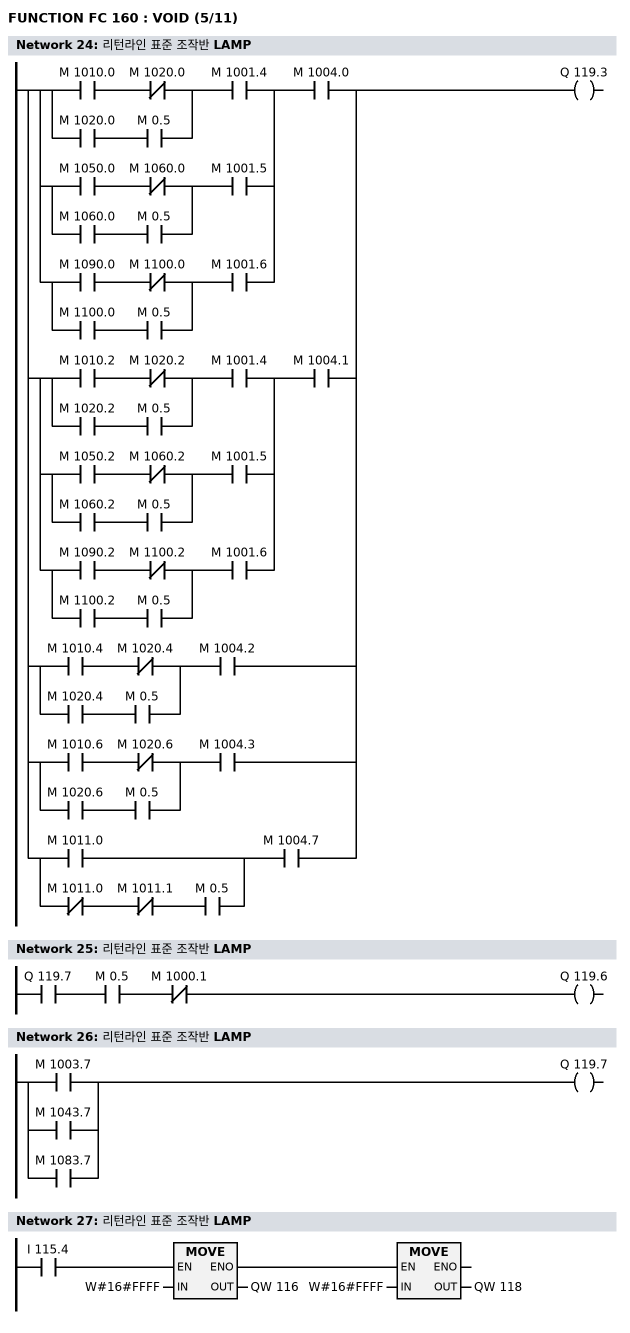

      A(    ;
      A(    ;
      A     M   1010.0;
      AN    M   1020.0;
      O     ;
      A     M   1020.0;
      A     M      0.5;
      )     ;
      A     M   1001.4;
      O     ;
      A(    ;
      A     M   1050.0;
      AN    M   1060.0;
      O     ;
      A     M   1060.0;
      A     M      0.5;
      )     ;
      A     M   1001.5;
      O     ;
      A(    ;
      A     M   1090.0;
      AN    M   1100.0;
      O     ;
      A     M   1100.0;
      A     M      0.5;
      )     ;
      A     M   1001.6;
      )     ;
      A     M   1004.0;
      O     ;
      A(    ;
      A(    ;
      A     M   1010.2;
      AN    M   1020.2;
      O     ;
      A     M   1020.2;
      A     M      0.5;
      )     ;
      A     M   1001.4;
      O     ;
      A(    ;
      A     M   1050.2;
      AN    M   1060.2;
      O     ;
      A     M   1060.2;
      A     M      0.5;
      )     ;
      A     M   1001.5;
      O     ;
      A(    ;
      A     M   1090.2;
      AN    M   1100.2;
      O     ;
      A     M   1100.2;
      A     M      0.5;
      )     ;
      A     M   1001.6;
      )     ;
      A     M   1004.1;
      O     ;
      A(    ;
      A     M   1010.4;
      AN    M   1020.4;
      O     ;
      A     M   1020.4;
      A     M      0.5;
      )     ;
      A     M   1004.2;
      O     ;
      A(    ;
      A     M   1010.6;
      AN    M   1020.6;
      O     ;
      A     M   1020.6;
      A     M      0.5;
      )     ;
      A     M   1004.3;
      O     ;
      A(    ;
      O     M   1011.0;
      O     ;
      AN    M   1011.0;
      AN    M   1011.1;
      A     M      0.5;
      )     ;
      A     M   1004.7;
      =     Q    119.3;
NETWORK
TITLE =리턴라인 표준 조작반 LAMP

      A     Q    119.7;
      A     M      0.5;
      AN    M   1000.1;
      =     Q    119.6;
NETWORK
TITLE =리턴라인 표준 조작반 LAMP

      O     M   1003.7;
      O     M   1043.7;
      O     M   1083.7;
      =     Q    119.7;
NETWORK
TITLE =리턴라인 표준 조작반 LAMP

      A(    ;
      A     I    115.4;
      JNB   _001;
      L     W#16#FFFF;
      T     QW   116;
      SET   ;
      SAVE  ;
      CLR   ;
_001: A     BR;
      )     ;
      JNB   _002;
      L     W#16#FFFF;
      T     QW   118;
_002: NOP   0;
NETWORK
TITLE =리턴라인 표준 조작반 LAMP
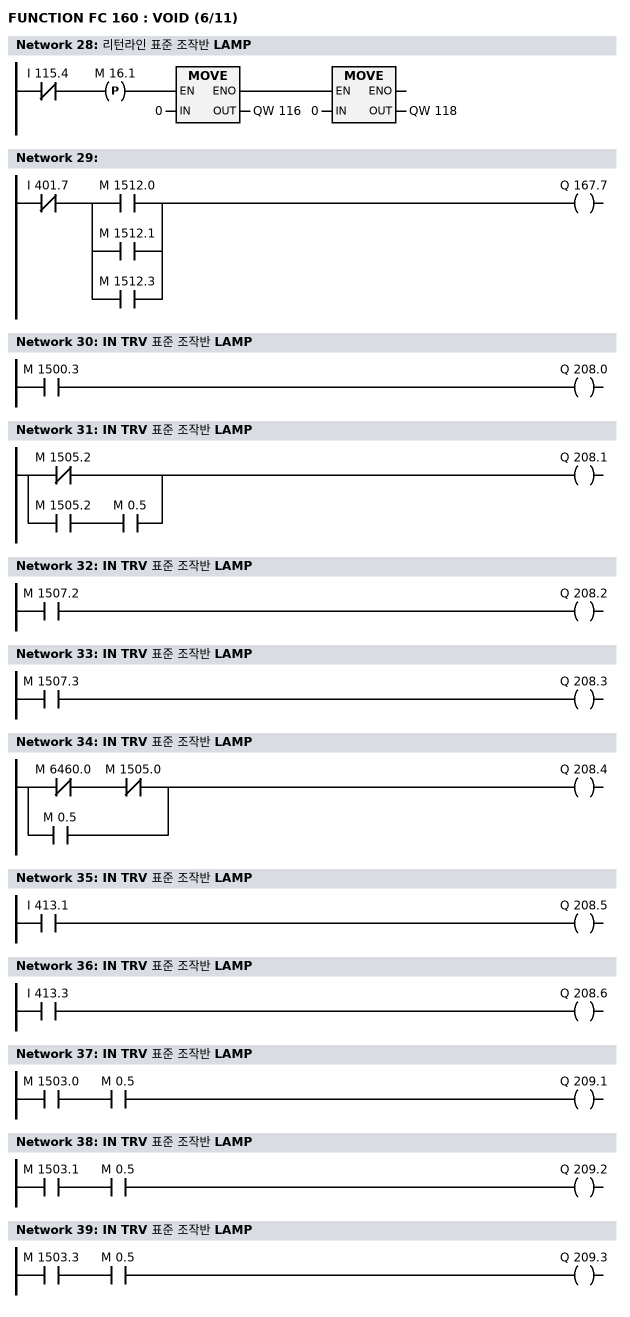

      A(    ;
      AN    I    115.4;
      FP    M     16.1;
      JNB   _003;
      L     0;
      T     QW   116;
      SET   ;
      SAVE  ;
      CLR   ;
_003: A     BR;
      )     ;
      JNB   _004;
      L     0;
      T     QW   118;
_004: NOP   0;
NETWORK
TITLE =

      AN    I    401.7;
      A(    ;
      O     M   1512.0;
      O     M   1512.1;
      O     M   1512.3;
      )     ;
      =     Q    167.7;
NETWORK
TITLE =IN TRV 표준 조작반 LAMP

      A     M   1500.3;
      =     Q    208.0;
NETWORK
TITLE =IN TRV 표준 조작반 LAMP

      ON    M   1505.2;
      O     ;
      A     M   1505.2;
      A     M      0.5;
      =     Q    208.1;
NETWORK
TITLE =IN TRV 표준 조작반 LAMP

      A     M   1507.2;
      =     Q    208.2;
NETWORK
TITLE =IN TRV 표준 조작반 LAMP

      A     M   1507.3;
      =     Q    208.3;
NETWORK
TITLE =IN TRV 표준 조작반 LAMP

      AN    M   6460.0;
      AN    M   1505.0;
      O     M      0.5;
      =     Q    208.4;
NETWORK
TITLE =IN TRV 표준 조작반 LAMP

      A     I    413.1;
      =     Q    208.5;
NETWORK
TITLE =IN TRV 표준 조작반 LAMP

      A     I    413.3;
      =     Q    208.6;
NETWORK
TITLE =IN TRV 표준 조작반 LAMP

      A     M   1503.0;
      A     M      0.5;
      =     Q    209.1;
NETWORK
TITLE =IN TRV 표준 조작반 LAMP

      A     M   1503.1;
      A     M      0.5;
      =     Q    209.2;
NETWORK
TITLE =IN TRV 표준 조작반 LAMP

      A     M   1503.3;
      A     M      0.5;
      =     Q    209.3;
NETWORK
TITLE =IN TRV 표준 조작반 LAMP
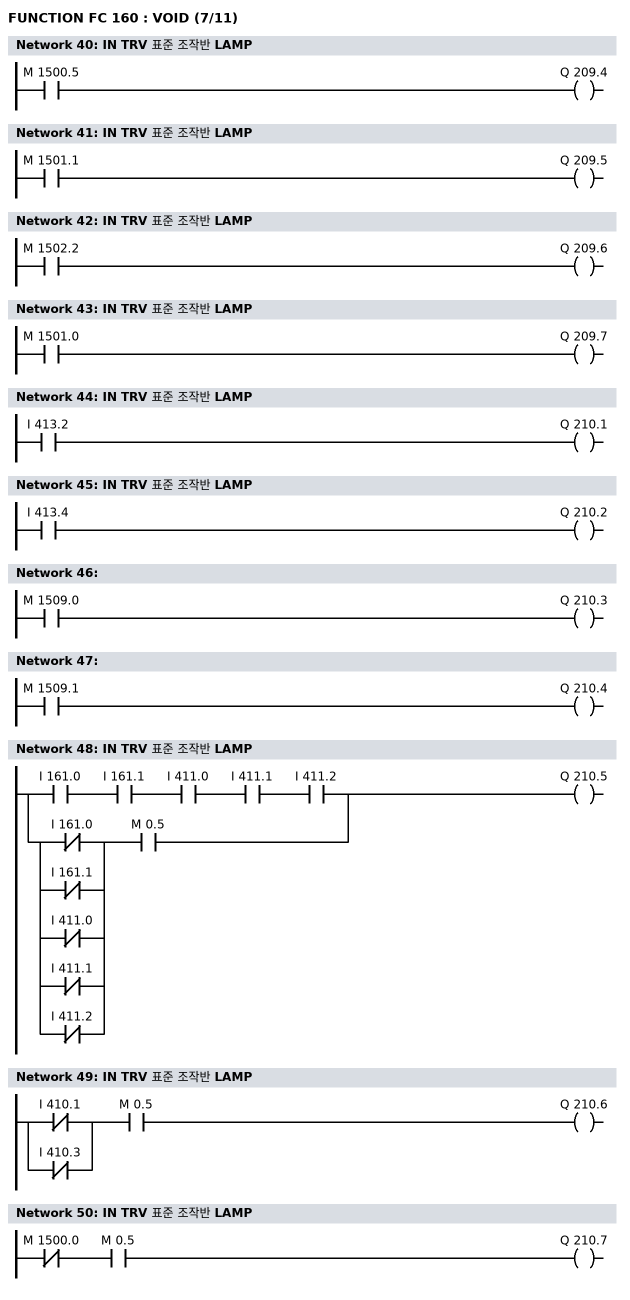

      A     M   1500.5;
      =     Q    209.4;
NETWORK
TITLE =IN TRV 표준 조작반 LAMP

      A     M   1501.1;
      =     Q    209.5;
NETWORK
TITLE =IN TRV 표준 조작반 LAMP

      A     M   1502.2;
      =     Q    209.6;
NETWORK
TITLE =IN TRV 표준 조작반 LAMP

      A     M   1501.0;
      =     Q    209.7;
NETWORK
TITLE =IN TRV 표준 조작반 LAMP

      A     I    413.2;
      =     Q    210.1;
NETWORK
TITLE =IN TRV 표준 조작반 LAMP

      A     I    413.4;
      =     Q    210.2;
NETWORK
TITLE =

      A     M   1509.0;
      =     Q    210.3;
NETWORK
TITLE =

      A     M   1509.1;
      =     Q    210.4;
NETWORK
TITLE =IN TRV 표준 조작반 LAMP

      A     I    161.0;
      A     I    161.1;
      A     I    411.0;
      A     I    411.1;
      A     I    411.2;
      O     ;
      A(    ;
      ON    I    161.0;
      ON    I    161.1;
      ON    I    411.0;
      ON    I    411.1;
      ON    I    411.2;
      )     ;
      A     M      0.5;
      =     Q    210.5;
NETWORK
TITLE =IN TRV 표준 조작반 LAMP

      A(    ;
      ON    I    410.1;
      ON    I    410.3;
      )     ;
      A     M      0.5;
      =     Q    210.6;
NETWORK
TITLE =IN TRV 표준 조작반 LAMP

      AN    M   1500.0;
      A     M      0.5;
      =     Q    210.7;
NETWORK
TITLE =IN TRV 표준 조작반 LAMP
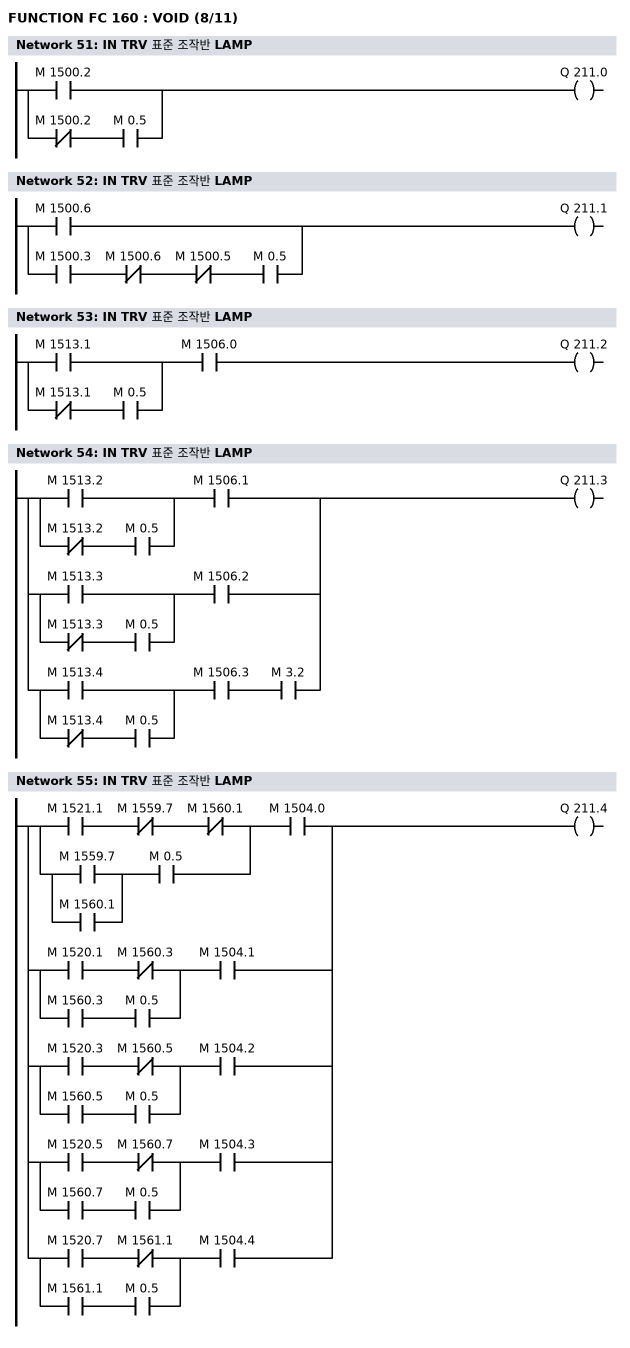

      O     M   1500.2;
      O     ;
      AN    M   1500.2;
      A     M      0.5;
      =     Q    211.0;
NETWORK
TITLE =IN TRV 표준 조작반 LAMP

      O     M   1500.6;
      O     ;
      A     M   1500.3;
      AN    M   1500.6;
      AN    M   1500.5;
      A     M      0.5;
      =     Q    211.1;
NETWORK
TITLE =IN TRV 표준 조작반 LAMP

      A(    ;
      O     M   1513.1;
      O     ;
      AN    M   1513.1;
      A     M      0.5;
      )     ;
      A     M   1506.0;
      =     Q    211.2;
NETWORK
TITLE =IN TRV 표준 조작반 LAMP

      A(    ;
      O     M   1513.2;
      O     ;
      AN    M   1513.2;
      A     M      0.5;
      )     ;
      A     M   1506.1;
      O     ;
      A(    ;
      O     M   1513.3;
      O     ;
      AN    M   1513.3;
      A     M      0.5;
      )     ;
      A     M   1506.2;
      O     ;
      A(    ;
      O     M   1513.4;
      O     ;
      AN    M   1513.4;
      A     M      0.5;
      )     ;
      A     M   1506.3;
      A     M      3.2;
      =     Q    211.3;
NETWORK
TITLE =IN TRV 표준 조작반 LAMP

      A(    ;
      A     M   1521.1;
      AN    M   1559.7;
      AN    M   1560.1;
      O     ;
      A(    ;
      O     M   1559.7;
      O     M   1560.1;
      )     ;
      A     M      0.5;
      )     ;
      A     M   1504.0;
      O     ;
      A(    ;
      A     M   1520.1;
      AN    M   1560.3;
      O     ;
      A     M   1560.3;
      A     M      0.5;
      )     ;
      A     M   1504.1;
      O     ;
      A(    ;
      A     M   1520.3;
      AN    M   1560.5;
      O     ;
      A     M   1560.5;
      A     M      0.5;
      )     ;
      A     M   1504.2;
      O     ;
      A(    ;
      A     M   1520.5;
      AN    M   1560.7;
      O     ;
      A     M   1560.7;
      A     M      0.5;
      )     ;
      A     M   1504.3;
      O     ;
      A(    ;
      A     M   1520.7;
      AN    M   1561.1;
      O     ;
      A     M   1561.1;
      A     M      0.5;
      )     ;
      A     M   1504.4;
      =     Q    211.4;
NETWORK
TITLE =IN TRV 표준 조작반 LAMP
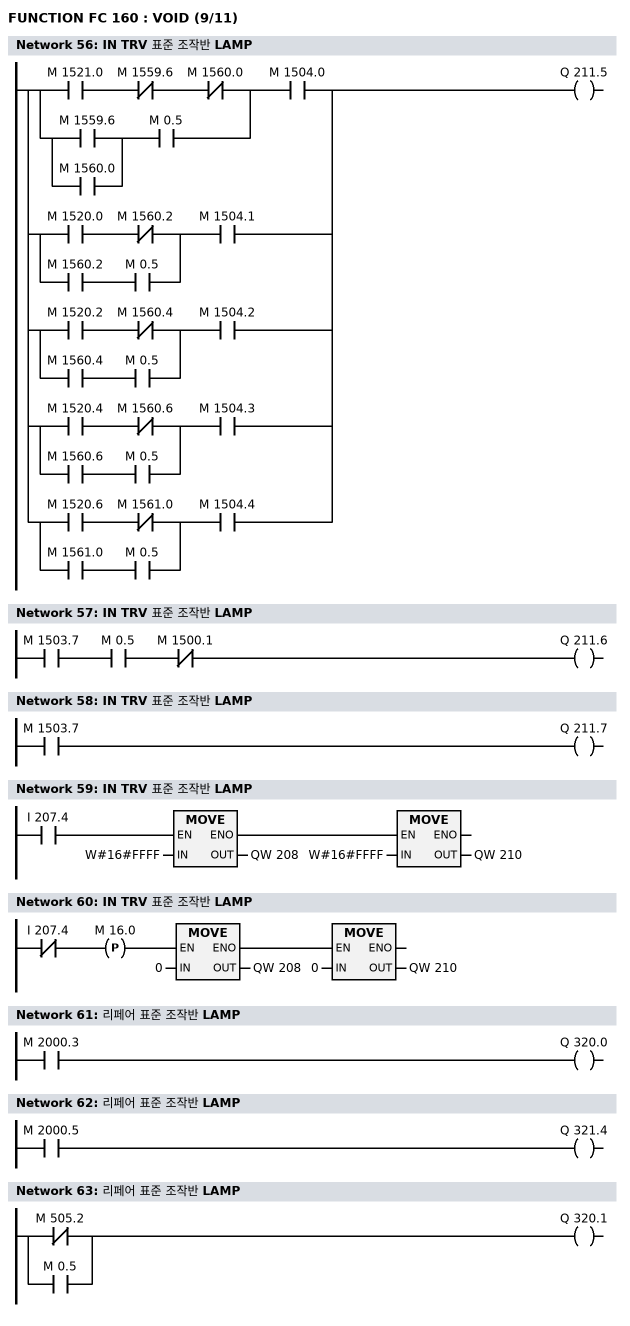

      A(    ;
      A     M   1521.0;
      AN    M   1559.6;
      AN    M   1560.0;
      O     ;
      A(    ;
      O     M   1559.6;
      O     M   1560.0;
      )     ;
      A     M      0.5;
      )     ;
      A     M   1504.0;
      O     ;
      A(    ;
      A     M   1520.0;
      AN    M   1560.2;
      O     ;
      A     M   1560.2;
      A     M      0.5;
      )     ;
      A     M   1504.1;
      O     ;
      A(    ;
      A     M   1520.2;
      AN    M   1560.4;
      O     ;
      A     M   1560.4;
      A     M      0.5;
      )     ;
      A     M   1504.2;
      O     ;
      A(    ;
      A     M   1520.4;
      AN    M   1560.6;
      O     ;
      A     M   1560.6;
      A     M      0.5;
      )     ;
      A     M   1504.3;
      O     ;
      A(    ;
      A     M   1520.6;
      AN    M   1561.0;
      O     ;
      A     M   1561.0;
      A     M      0.5;
      )     ;
      A     M   1504.4;
      =     Q    211.5;
NETWORK
TITLE =IN TRV 표준 조작반 LAMP

      A     M   1503.7;
      A     M      0.5;
      AN    M   1500.1;
      =     Q    211.6;
NETWORK
TITLE =IN TRV 표준 조작반 LAMP

      A     M   1503.7;
      =     Q    211.7;
NETWORK
TITLE =IN TRV 표준 조작반 LAMP

      A(    ;
      A     I    207.4;
      JNB   _005;
      L     W#16#FFFF;
      T     QW   208;
      SET   ;
      SAVE  ;
      CLR   ;
_005: A     BR;
      )     ;
      JNB   _006;
      L     W#16#FFFF;
      T     QW   210;
_006: NOP   0;
NETWORK
TITLE =IN TRV 표준 조작반 LAMP

      A(    ;
      AN    I    207.4;
      FP    M     16.0;
      JNB   _007;
      L     0;
      T     QW   208;
      SET   ;
      SAVE  ;
      CLR   ;
_007: A     BR;
      )     ;
      JNB   _008;
      L     0;
      T     QW   210;
_008: NOP   0;
NETWORK
TITLE =리페어 표준 조작반 LAMP

      A     M   2000.3;
      =     Q    320.0;
NETWORK
TITLE =리페어 표준 조작반 LAMP

      A     M   2000.5;
      =     Q    321.4;
NETWORK
TITLE =리페어 표준 조작반 LAMP

      ON    M    505.2;
      O     M      0.5;
      =     Q    320.1;
NETWORK
TITLE =리페어 표준 조작반 LAMP
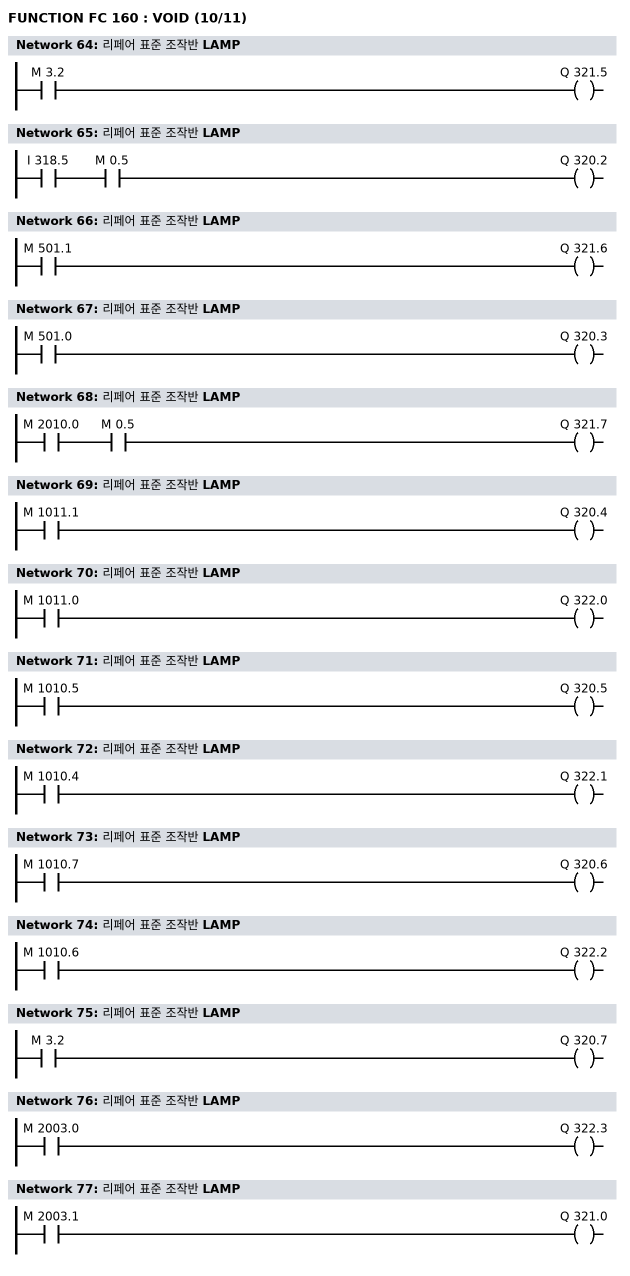

      A     M      3.2;
      =     Q    321.5;
NETWORK
TITLE =리페어 표준 조작반 LAMP

      A     I    318.5;
      A     M      0.5;
      =     Q    320.2;
NETWORK
TITLE =리페어 표준 조작반 LAMP

      A     M    501.1;
      =     Q    321.6;
NETWORK
TITLE =리페어 표준 조작반 LAMP

      A     M    501.0;
      =     Q    320.3;
NETWORK
TITLE =리페어 표준 조작반 LAMP

      A     M   2010.0;
      A     M      0.5;
      =     Q    321.7;
NETWORK
TITLE =리페어 표준 조작반 LAMP

      A     M   1011.1;
      =     Q    320.4;
NETWORK
TITLE =리페어 표준 조작반 LAMP

      A     M   1011.0;
      =     Q    322.0;
NETWORK
TITLE =리페어 표준 조작반 LAMP

      A     M   1010.5;
      =     Q    320.5;
NETWORK
TITLE =리페어 표준 조작반 LAMP

      A     M   1010.4;
      =     Q    322.1;
NETWORK
TITLE =리페어 표준 조작반 LAMP

      A     M   1010.7;
      =     Q    320.6;
NETWORK
TITLE =리페어 표준 조작반 LAMP

      A     M   1010.6;
      =     Q    322.2;
NETWORK
TITLE =리페어 표준 조작반 LAMP

      A     M      3.2;
      =     Q    320.7;
NETWORK
TITLE =리페어 표준 조작반 LAMP

      A     M   2003.0;
      =     Q    322.3;
NETWORK
TITLE =리페어 표준 조작반 LAMP

      A     M   2003.1;
      =     Q    321.0;
NETWORK
TITLE =리페어 표준 조작반 LAMP
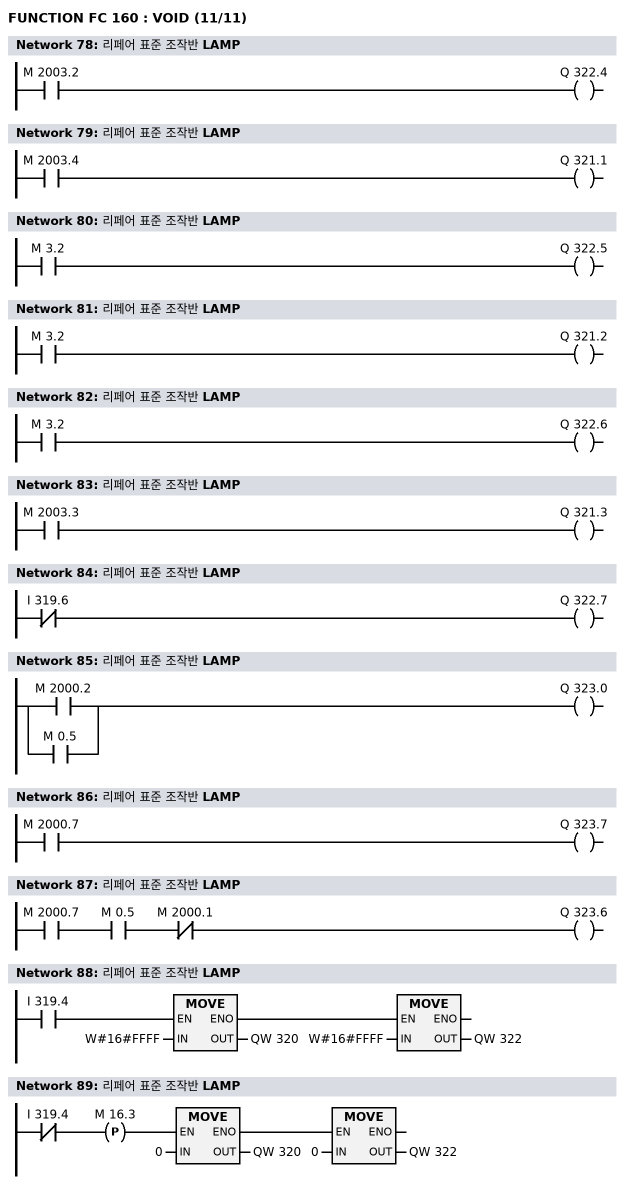

      A     M   2003.2;
      =     Q    322.4;
NETWORK
TITLE =리페어 표준 조작반 LAMP

      A     M   2003.4;
      =     Q    321.1;
NETWORK
TITLE =리페어 표준 조작반 LAMP

      A     M      3.2;
      =     Q    322.5;
NETWORK
TITLE =리페어 표준 조작반 LAMP

      A     M      3.2;
      =     Q    321.2;
NETWORK
TITLE =리페어 표준 조작반 LAMP

      A     M      3.2;
      =     Q    322.6;
NETWORK
TITLE =리페어 표준 조작반 LAMP

      A     M   2003.3;
      =     Q    321.3;
NETWORK
TITLE =리페어 표준 조작반 LAMP

      AN    I    319.6;
      =     Q    322.7;
NETWORK
TITLE =리페어 표준 조작반 LAMP

      O     M   2000.2;
      O     M      0.5;
      =     Q    323.0;
NETWORK
TITLE =리페어 표준 조작반 LAMP

      A     M   2000.7;
      =     Q    323.7;
NETWORK
TITLE =리페어 표준 조작반 LAMP

      A     M   2000.7;
      A     M      0.5;
      AN    M   2000.1;
      =     Q    323.6;
NETWORK
TITLE =리페어 표준 조작반 LAMP

      A(    ;
      A     I    319.4;
      JNB   _009;
      L     W#16#FFFF;
      T     QW   320;
      SET   ;
      SAVE  ;
      CLR   ;
_009: A     BR;
      )     ;
      JNB   _00a;
      L     W#16#FFFF;
      T     QW   322;
_00a: NOP   0;
NETWORK
TITLE =리페어 표준 조작반 LAMP

      A(    ;
      AN    I    319.4;
      FP    M     16.3;
      JNB   _00b;
      L     0;
      T     QW   320;
      SET   ;
      SAVE  ;
      CLR   ;
_00b: A     BR;
      )     ;
      JNB   _00c;
      L     0;
      T     QW   322;
_00c: NOP   0;
END_FUNCTION

FUNCTION FC 324 : VOID
TITLE =
VERSION : 0.1

BEGIN
NETWORK
TITLE =
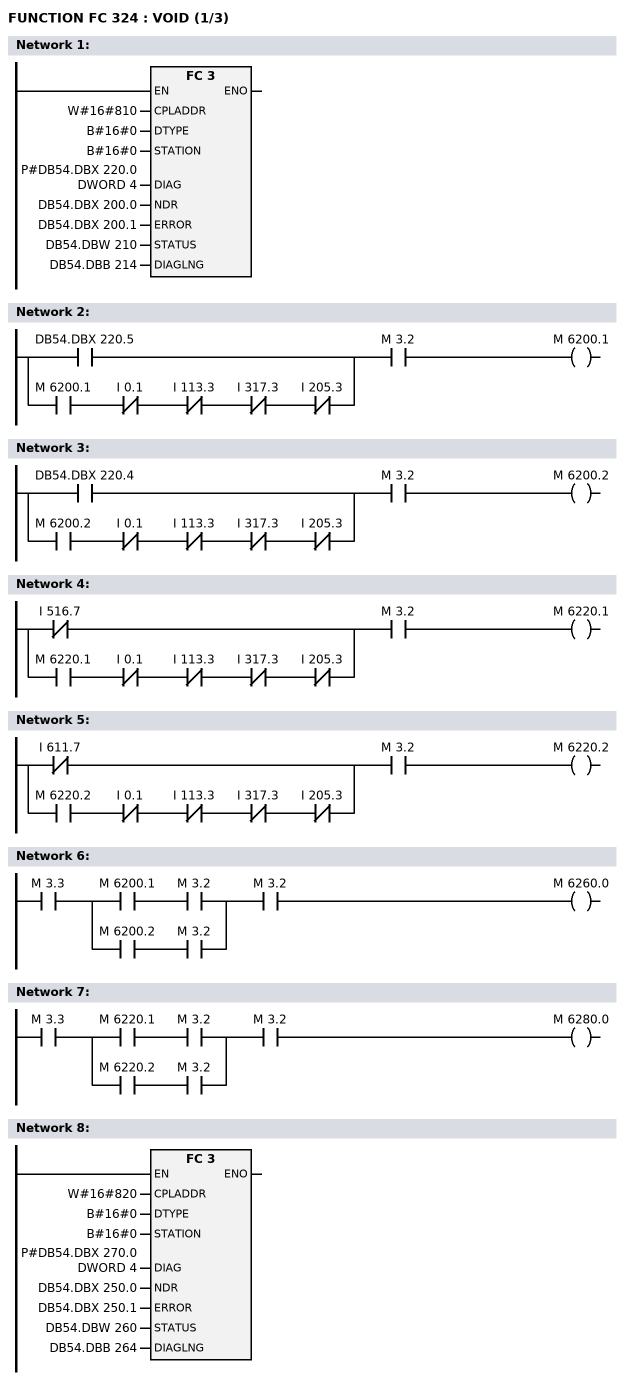

      CALL FC     3 (
           CPLADDR                  := W#16#810,
           DTYPE                    := B#16#0,
           STATION                  := B#16#0,
           DIAG                     := P#DB54.DBX 220.0 DWORD 4,
           NDR                      := DB54.DBX  200.0,
           ERROR                    := DB54.DBX  200.1,
           STATUS                   := DB54.DBW  210,
           DIAGLNG                  := DB54.DBB  214);
      NOP   0;
NETWORK
TITLE =

      A(    ;
      O     DB54.DBX  220.5;
      O     ;
      A     M   6200.1;
      AN    I      0.1;
      AN    I    113.3;
      AN    I    317.3;
      AN    I    205.3;
      )     ;
      A     M      3.2;
      =     M   6200.1;
NETWORK
TITLE =

      A(    ;
      O     DB54.DBX  220.4;
      O     ;
      A     M   6200.2;
      AN    I      0.1;
      AN    I    113.3;
      AN    I    317.3;
      AN    I    205.3;
      )     ;
      A     M      3.2;
      =     M   6200.2;
NETWORK
TITLE =

      A(    ;
      ON    I    516.7;
      O     ;
      A     M   6220.1;
      AN    I      0.1;
      AN    I    113.3;
      AN    I    317.3;
      AN    I    205.3;
      )     ;
      A     M      3.2;
      =     M   6220.1;
NETWORK
TITLE =

      A(    ;
      ON    I    611.7;
      O     ;
      A     M   6220.2;
      AN    I      0.1;
      AN    I    113.3;
      AN    I    317.3;
      AN    I    205.3;
      )     ;
      A     M      3.2;
      =     M   6220.2;
NETWORK
TITLE =

      A     M      3.3;
      A(    ;
      A     M   6200.1;
      A     M      3.2;
      O     ;
      A     M   6200.2;
      A     M      3.2;
      )     ;
      A     M      3.2;
      =     M   6260.0;
NETWORK
TITLE =

      A     M      3.3;
      A(    ;
      A     M   6220.1;
      A     M      3.2;
      O     ;
      A     M   6220.2;
      A     M      3.2;
      )     ;
      A     M      3.2;
      =     M   6280.0;
NETWORK
TITLE =

      CALL FC     3 (
           CPLADDR                  := W#16#820,
           DTYPE                    := B#16#0,
           STATION                  := B#16#0,
           DIAG                     := P#DB54.DBX 270.0 DWORD 4,
           NDR                      := DB54.DBX  250.0,
           ERROR                    := DB54.DBX  250.1,
           STATUS                   := DB54.DBW  260,
           DIAGLNG                  := DB54.DBB  264);
      NOP   0;
NETWORK
TITLE =
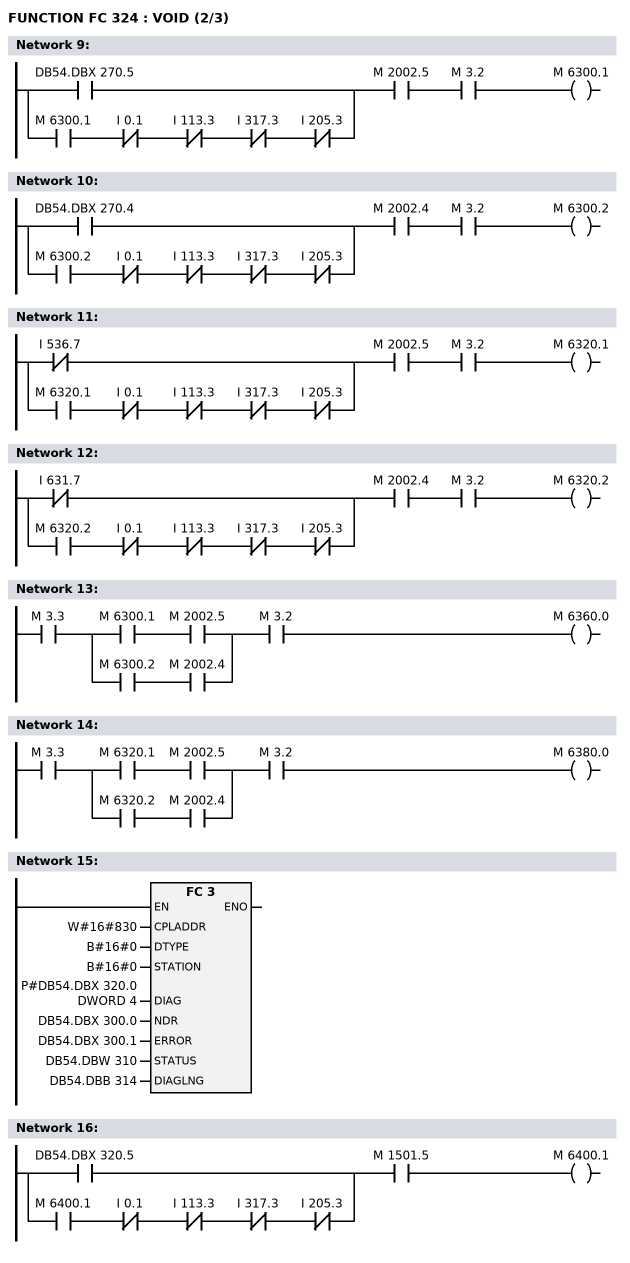

      A(    ;
      O     DB54.DBX  270.5;
      O     ;
      A     M   6300.1;
      AN    I      0.1;
      AN    I    113.3;
      AN    I    317.3;
      AN    I    205.3;
      )     ;
      A     M   2002.5;
      A     M      3.2;
      =     M   6300.1;
NETWORK
TITLE =

      A(    ;
      O     DB54.DBX  270.4;
      O     ;
      A     M   6300.2;
      AN    I      0.1;
      AN    I    113.3;
      AN    I    317.3;
      AN    I    205.3;
      )     ;
      A     M   2002.4;
      A     M      3.2;
      =     M   6300.2;
NETWORK
TITLE =

      A(    ;
      ON    I    536.7;
      O     ;
      A     M   6320.1;
      AN    I      0.1;
      AN    I    113.3;
      AN    I    317.3;
      AN    I    205.3;
      )     ;
      A     M   2002.5;
      A     M      3.2;
      =     M   6320.1;
NETWORK
TITLE =

      A(    ;
      ON    I    631.7;
      O     ;
      A     M   6320.2;
      AN    I      0.1;
      AN    I    113.3;
      AN    I    317.3;
      AN    I    205.3;
      )     ;
      A     M   2002.4;
      A     M      3.2;
      =     M   6320.2;
NETWORK
TITLE =

      A     M      3.3;
      A(    ;
      A     M   6300.1;
      A     M   2002.5;
      O     ;
      A     M   6300.2;
      A     M   2002.4;
      )     ;
      A     M      3.2;
      =     M   6360.0;
NETWORK
TITLE =

      A     M      3.3;
      A(    ;
      A     M   6320.1;
      A     M   2002.5;
      O     ;
      A     M   6320.2;
      A     M   2002.4;
      )     ;
      A     M      3.2;
      =     M   6380.0;
NETWORK
TITLE =

      CALL FC     3 (
           CPLADDR                  := W#16#830,
           DTYPE                    := B#16#0,
           STATION                  := B#16#0,
           DIAG                     := P#DB54.DBX 320.0 DWORD 4,
           NDR                      := DB54.DBX  300.0,
           ERROR                    := DB54.DBX  300.1,
           STATUS                   := DB54.DBW  310,
           DIAGLNG                  := DB54.DBB  314);
      NOP   0;
NETWORK
TITLE =

      A(    ;
      O     DB54.DBX  320.5;
      O     ;
      A     M   6400.1;
      AN    I      0.1;
      AN    I    113.3;
      AN    I    317.3;
      AN    I    205.3;
      )     ;
      A     M   1501.5;
      =     M   6400.1;
NETWORK
TITLE =
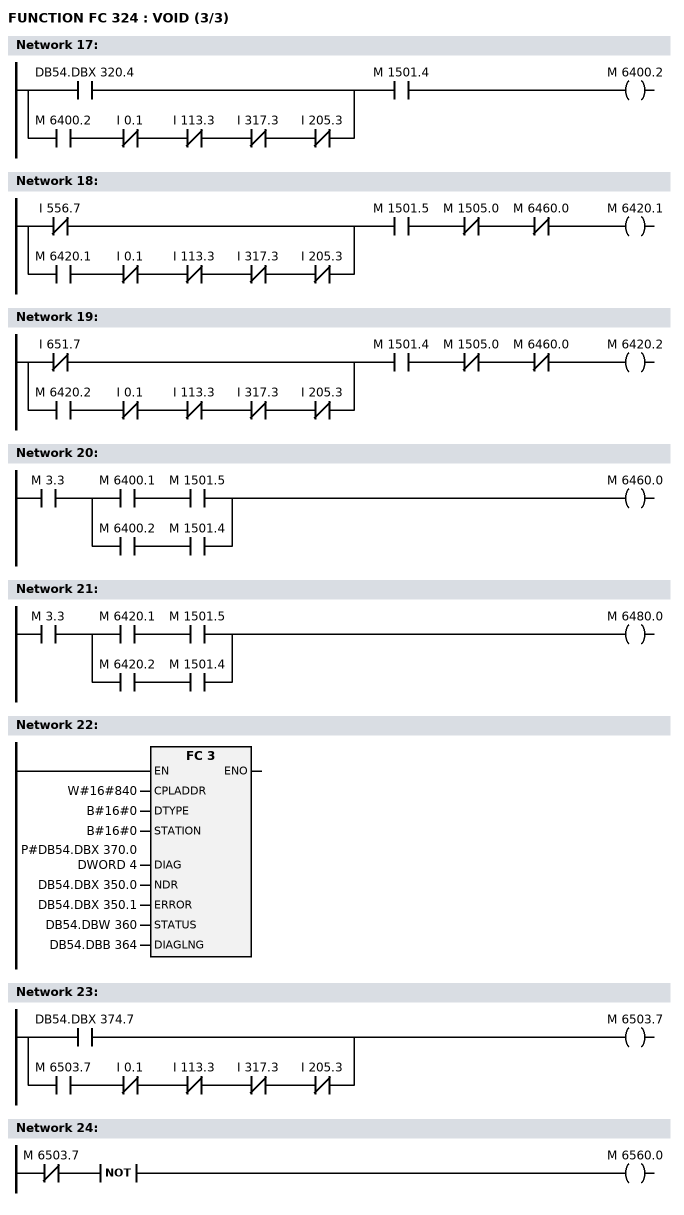

      A(    ;
      O     DB54.DBX  320.4;
      O     ;
      A     M   6400.2;
      AN    I      0.1;
      AN    I    113.3;
      AN    I    317.3;
      AN    I    205.3;
      )     ;
      A     M   1501.4;
      =     M   6400.2;
NETWORK
TITLE =

      A(    ;
      ON    I    556.7;
      O     ;
      A     M   6420.1;
      AN    I      0.1;
      AN    I    113.3;
      AN    I    317.3;
      AN    I    205.3;
      )     ;
      A     M   1501.5;
      AN    M   1505.0;
      AN    M   6460.0;
      =     M   6420.1;
NETWORK
TITLE =

      A(    ;
      ON    I    651.7;
      O     ;
      A     M   6420.2;
      AN    I      0.1;
      AN    I    113.3;
      AN    I    317.3;
      AN    I    205.3;
      )     ;
      A     M   1501.4;
      AN    M   1505.0;
      AN    M   6460.0;
      =     M   6420.2;
NETWORK
TITLE =

      A     M      3.3;
      A(    ;
      A     M   6400.1;
      A     M   1501.5;
      O     ;
      A     M   6400.2;
      A     M   1501.4;
      )     ;
      =     M   6460.0;
NETWORK
TITLE =

      A     M      3.3;
      A(    ;
      A     M   6420.1;
      A     M   1501.5;
      O     ;
      A     M   6420.2;
      A     M   1501.4;
      )     ;
      =     M   6480.0;
NETWORK
TITLE =

      CALL FC     3 (
           CPLADDR                  := W#16#840,
           DTYPE                    := B#16#0,
           STATION                  := B#16#0,
           DIAG                     := P#DB54.DBX 370.0 DWORD 4,
           NDR                      := DB54.DBX  350.0,
           ERROR                    := DB54.DBX  350.1,
           STATUS                   := DB54.DBW  360,
           DIAGLNG                  := DB54.DBB  364);
      NOP   0;
NETWORK
TITLE =

      O     DB54.DBX  374.7;
      O     ;
      A     M   6503.7;
      AN    I      0.1;
      AN    I    113.3;
      AN    I    317.3;
      AN    I    205.3;
      =     M   6503.7;
NETWORK
TITLE =

      AN    M   6503.7;
      NOT   ;
      =     M   6560.0;
END_FUNCTION

FUNCTION_BLOCK FB 406
TITLE =Data Block Move Program
AUTHOR : HMC
FAMILY : Car_Type
NAME : Car_Type
VERSION : 1.0


VAR_INPUT
  FWD_Pulse : BOOL ;
  RET_Pulse : BOOL ;
  Source_DB : INT ;
  Start_Add : INT ;
  Stn_Amount : INT ;
  Byte_per_Stn : INT ;
  Cpu_Run_Pulse : BOOL ;
END_VAR
VAR_OUTPUT
  Complete : BOOL ;
END_VAR
VAR
  Operation : BOOL ;
  Mask_Arr : ARRAY  [0 .. 599 ] OF BYTE ;
  Ret : INT ;
  Data_Type : WORD ;
  Data_Length : INT ;
  Secend_Stn_Add : INT ;
  Fill_Source : WORD ;
END_VAR
VAR_TEMP
  First_Stn : ANY ;
  Mask : ANY ;
  Second_Stn : ANY ;
  Save_AR1 : DWORD ;
  Save_AR2 : DWORD ;
  Save_DB : INT ;
  Save_DI : INT ;
  First_Stn_1 : ANY ;
END_VAR
BEGIN
NETWORK
TITLE =Save adress register and DB's

      TAR1  #Save_AR1; // Save adress register 1
      TAR2  #Save_AR2; // Save adress register 2
      L     DBNO; // loads the number of the shared open data block
      T     #Save_DB;
      L     DINO; // loads the number of the opened instance data block
      T     #Save_DI;
NETWORK
TITLE =Operation Pulse

      O     #FWD_Pulse; // External ForwardOperation Signal
      O     #RET_Pulse; // External Return Operation Signal
      FP    #Operation; // Operation Pulse
      JNB   _End; // Jump to End
NETWORK
TITLE =Data Type Select In ANY Type Parameter

      A(    ; // If Source DB is Not Zero
      L     #Source_DB;
      L     0;
      <>I   ;
      )     ;
      JNB   _001; // Jump to Next Step
      L     W#16#8400; // Load "8400" _ Means "DB Area"
      T     #Data_Type; // Transfer to Data_Type
_001: NOP   0;
NETWORK
TITLE =Data Type Select In ANY Type Parameter

      A(    ; // If DB_NO is Zero
      L     #Source_DB;
      L     0;
      ==I   ;
      )     ;
      JNB   _002; // Jump to Next Step
      L     W#16#8300; // Load "8300" _ Means "Bit Memory Area"
      T     #Data_Type; // Transfer to Data_Type
_002: NOP   0;
NETWORK
TITLE =Data Length Select

      L     #Stn_Amount; // Station Amount - 1
      L     1;
      -I    ;
      L     #Byte_per_Stn; // Multi Length Per Station
      *I    ;
      T     #Data_Length; // Transfer to Data Length
NETWORK
TITLE =2nd Station Address Select

      L     #Start_Add; // Pluse Start Address And Length
      L     #Byte_per_Stn;
      +I    ;
      T     #Secend_Stn_Add; // Transfer to Second Station Address
NETWORK
TITLE =Make a "ANY" Type Data

      LAR1  P##First_Stn; // Load 1st Station Address of ANY Pointer In "AR1"

      L     B#16#10; // Load Syntax ID For S7 "10"
      T     LB [AR1,P#0.0]; // Transfer ID to the ANY Pointer

      L     B#16#2; // Load Data Type _ "2" means "BYTE"
      T     LB [AR1,P#1.0]; // Transfer Data Type to the ANY Pointer

      L     #Data_Length; // Load the Length of Source Data
      T     LW [AR1,P#2.0]; // Transfer the Numbers to the ANY Pointer

      L     #Source_DB; // Load DB Number _ "0" means don't use "DB"
      T     LW [AR1,P#4.0]; // Transfer the Numbers to the ANY Pointer

      L     #Data_Type; // Load Data Type _ "83" means "Bit Memory" Area
      T     LW [AR1,P#6.0]; //                  "84" means "DB" Area

      L     #Start_Add; // Load Start Address
      SLW   3; // Shift Left Word _ "3" Bit
      T     LW [AR1,P#8.0]; // Transfer the Address to the ANY Pointer

      LAR1  P##Mask; // Load 2nd Station Address of ANY Pointer In "AR1"

      L     B#16#10; //Load Syntax ID For S7 "10"
      T     LB [AR1,P#0.0]; //Load Syntax ID For S7 "10"

      L     B#16#2; //  Load Data Type _ "2" means "BYTE"
      T     LB [AR1,P#1.0]; // Transfer Data Type to the ANY Pointer

      L     #Data_Length; // Load the Length of Target Data
      T     LW [AR1,P#2.0]; // Transfer the Numbers to the ANY Pointer

      L     #Save_DI; // Load DB Number _ "0" means don't use "DB"
      T     LW [AR1,P#4.0]; // Transfer the Numbers to the ANY Pointer

      L     #Data_Type; // Load Data Type _ "83" means "Bit Memory" Area
      T     LW [AR1,P#6.0]; //                  "84" means "DB" Area

      L     16; //  Load Start Address
      SLW   3; // Shift Left Word _ "3" Bit
      T     LW [AR1,P#8.0]; // Transfer the Address to the ANY Pointer

NETWORK
TITLE =Make a "ANY" Type Data

      LAR1  P##Second_Stn; // Load 1st Station Address of ANY Pointer In "AR1"

      L     B#16#10; // Load Syntax ID For S7 "10"
      T     LB [AR1,P#0.0]; // Transfer ID to the ANY Pointer

      L     B#16#2; // Load Data Type _ "2" means "BYTE"
      T     LB [AR1,P#1.0]; // Transfer Data Type to the ANY Pointer

      L     #Data_Length; // Load the Length of Source Data
      T     LW [AR1,P#2.0]; // Transfer the Numbers to the ANY Pointer

      L     #Source_DB; // Load DB Number _ "0" means don't use "DB"
      T     LW [AR1,P#4.0]; // Transfer the Numbers to the ANY Pointer

      L     #Data_Type; // Load Data Type _ "83" means "Bit Memory" Area
      T     LW [AR1,P#6.0]; //                  "84" means "DB" Area

      L     #Secend_Stn_Add; // Load Second Station Address
      SLW   3; // Shift Left Word _ "3" Bit
      T     LW [AR1,P#8.0]; // Transfer the Address to the ANY Pointer
NETWORK
TITLE =Reset Car Type Transfer Complete Signal

      O     #FWD_Pulse; // External Forward Operation Signal
      O     #RET_Pulse; // External Return Operation Signal
      R     #Complete; // Reset Complete Signal
NETWORK
TITLE =Make Fill Source Data

      L     0;
      T     #Fill_Source;
NETWORK
TITLE =Fwd Block Move to Mask Area

      A     #FWD_Pulse; // External Forward Operation Signal
      AN    #Complete; // Complete Signal is False
      AN    #Cpu_Run_Pulse;
      JNB   _FWD;
      CALL SFC   20 (
           SRCBLK                   := #First_Stn,
           RET_VAL                  := #Ret,
           DSTBLK                   := #Mask);

NETWORK
TITLE =Clear Source Data Area


      CALL SFC   21 (
           IN0                      := #Fill_Source,// "Zero"
           RET_VAL                  := #Ret,
           OUT1                     := #First_Stn);// Transfer to First Station Area

NETWORK
TITLE =Fwd Block Move to Second Station Area


      CALL SFC   20 (
           SRCBLK                   := #Mask,
           RET_VAL                  := #Ret,
           DSTBLK                   := #Second_Stn);

NETWORK
TITLE =Clear Mask Data Area


      CALL SFC   21 (
           IN0                      := #Fill_Source,// "Zero"
           RET_VAL                  := #Ret,
           OUT1                     := #Mask);// Transfer to Mask Area
_FWD: NOP   0;
NETWORK
TITLE =Rev Block Move to Mask Area

      A     #RET_Pulse; // External Return Operation Signal
      AN    #Complete; // Complete Signal is False
      AN    #Cpu_Run_Pulse;
      JNB   _REV;
      CALL SFC   20 (
           SRCBLK                   := #Second_Stn,
           RET_VAL                  := #Ret,
           DSTBLK                   := #Mask);

NETWORK
TITLE =Clear Source Data Area


      CALL SFC   21 (
           IN0                      := #Fill_Source,// "Zero"
           RET_VAL                  := #Ret,
           OUT1                     := #Second_Stn);// Transfer to Second Station Area

NETWORK
TITLE =Rev Block Move to First Station Area


      CALL SFC   20 (
           SRCBLK                   := #Mask,
           RET_VAL                  := #Ret,
           DSTBLK                   := #First_Stn);

NETWORK
TITLE =Clear Mask Data Area


      CALL SFC   21 (
           IN0                      := #Fill_Source,// "Zero"
           RET_VAL                  := #Ret,
           OUT1                     := #Mask);// Transfer to Mask Area
_REV: NOP   0;
NETWORK
TITLE =Set Complete Signal

      S     #Complete;
_End: NOP   0;
END_FUNCTION_BLOCK

FUNCTION_BLOCK FB 426
TITLE =Sensor Error,Lamp Variables Program
AUTHOR : HMC
FAMILY : Common
NAME : Common
VERSION : 1.0


VAR_INPUT
  Enable_Aux : BOOL ;
  Adv_Amount : INT ;
  Ret_Amount : INT ;
  LS_Adv1 : BOOL ;
  LS_Ret1 : BOOL ;
  LS_Adv2 : BOOL ;
  LS_Ret2 : BOOL ;
  LS_Adv3 : BOOL ;
  LS_Ret3 : BOOL ;
  LS_Adv4 : BOOL ;
  LS_Ret4 : BOOL ;
  LS_Adv5 : BOOL ;
  LS_Ret5 : BOOL ;
  LS_Adv6 : BOOL ;
  LS_Ret6 : BOOL ;
  LS_Adv7 : BOOL ;
  LS_Ret7 : BOOL ;
  LS_Adv8 : BOOL ;
  LS_Ret8 : BOOL ;
  SOL_Adv : BOOL ;
  SOL_Ret : BOOL ;
  M_Ready : BOOL ;
  T_CHK1 : TIME ;
  T_CHK2 : TIME ;
  PB_Lamp_CHK : BOOL ;
  PB_Error_Rst : BOOL ;
  M_FLICK : BOOL ;
END_VAR
VAR_OUTPUT
  M_Adv_Err : BOOL ;
  M_Ret_Err : BOOL ;
  LP_Adv : BOOL ;
  LP_Ret : BOOL ;
  Visu_Adv : WORD ;
  Visu_Ret : WORD ;
END_VAR
VAR
  Error_T1 : SFB 4;
  Error_T2 : SFB 4;
  Adv_End_Aux : BOOL ;
  Ret_End_Aux : BOOL ;
  CHK_Aux1 : BOOL ;
  CHK_Aux2 : BOOL ;
  Error_T1_DN : BOOL ;
  Error_T2_DN : BOOL ;
  Adv_Memo : BOOL ;
  Visu_Adv_Arr : ARRAY  [0 .. 15 ] OF BOOL ;
  Visu_Ret_Arr : ARRAY  [0 .. 15 ] OF BOOL ;
  BLK_Move_Ret : INT ;
  Enable : BOOL ;
  Adv_End : BOOL ;
  Ret_End : BOOL ;
END_VAR
BEGIN
NETWORK
TITLE =
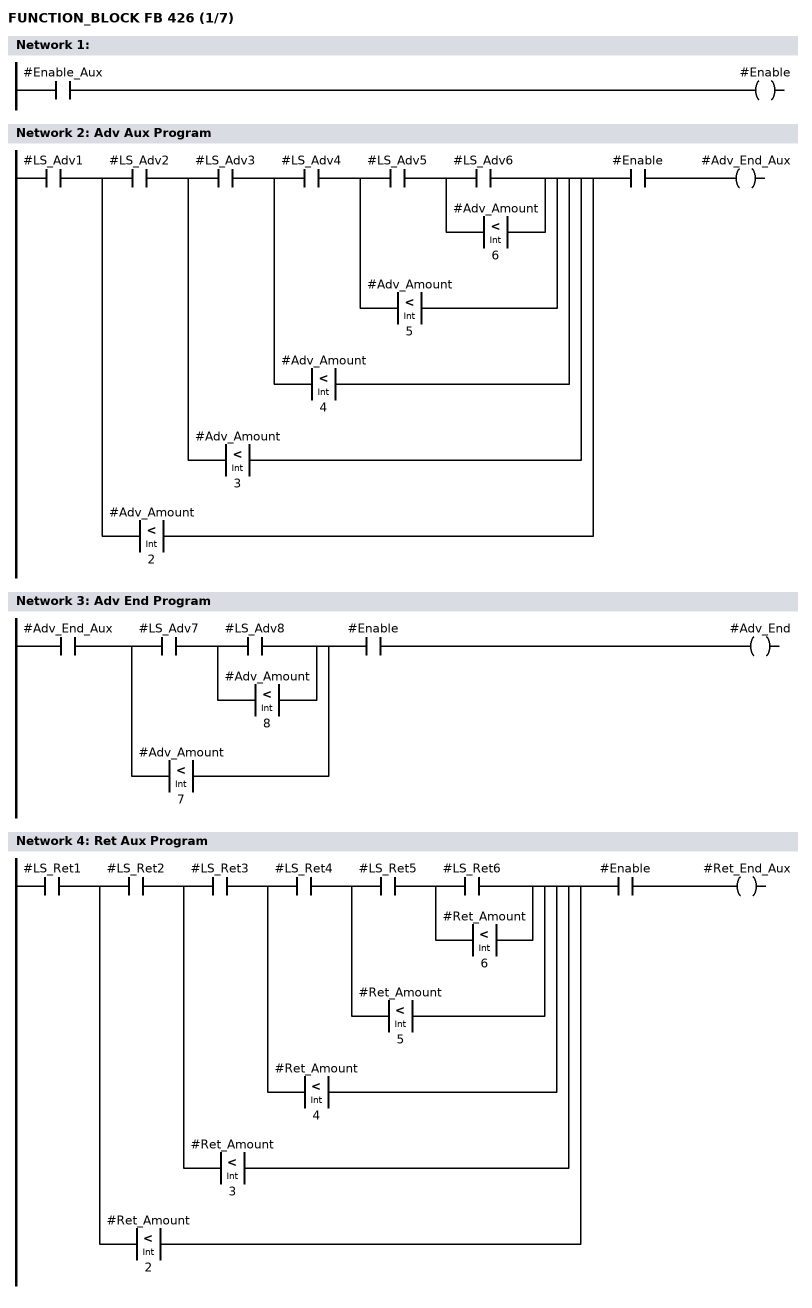

      A     #Enable_Aux;
      =     #Enable;
NETWORK
TITLE =Adv Aux Program

      A     #LS_Adv1;
      A(    ;
      A     #LS_Adv2;
      A(    ;
      A     #LS_Adv3;
      A(    ;
      A     #LS_Adv4;
      A(    ;
      A     #LS_Adv5;
      A(    ;
      O     #LS_Adv6;
      O(    ;
      L     #Adv_Amount;
      L     6;
      <I    ;
      )     ;
      )     ;
      O(    ;
      L     #Adv_Amount;
      L     5;
      <I    ;
      )     ;
      )     ;
      O(    ;
      L     #Adv_Amount;
      L     4;
      <I    ;
      )     ;
      )     ;
      O(    ;
      L     #Adv_Amount;
      L     3;
      <I    ;
      )     ;
      )     ;
      O(    ;
      L     #Adv_Amount;
      L     2;
      <I    ;
      )     ;
      )     ;
      A     #Enable;
      =     #Adv_End_Aux;
NETWORK
TITLE =Adv End Program

      A     #Adv_End_Aux;
      A(    ;
      A     #LS_Adv7;
      A(    ;
      O     #LS_Adv8;
      O(    ;
      L     #Adv_Amount;
      L     8;
      <I    ;
      )     ;
      )     ;
      O(    ;
      L     #Adv_Amount;
      L     7;
      <I    ;
      )     ;
      )     ;
      A     #Enable;
      =     #Adv_End;
NETWORK
TITLE =Ret Aux Program

      A     #LS_Ret1;
      A(    ;
      A     #LS_Ret2;
      A(    ;
      A     #LS_Ret3;
      A(    ;
      A     #LS_Ret4;
      A(    ;
      A     #LS_Ret5;
      A(    ;
      O     #LS_Ret6;
      O(    ;
      L     #Ret_Amount;
      L     6;
      <I    ;
      )     ;
      )     ;
      O(    ;
      L     #Ret_Amount;
      L     5;
      <I    ;
      )     ;
      )     ;
      O(    ;
      L     #Ret_Amount;
      L     4;
      <I    ;
      )     ;
      )     ;
      O(    ;
      L     #Ret_Amount;
      L     3;
      <I    ;
      )     ;
      )     ;
      O(    ;
      L     #Ret_Amount;
      L     2;
      <I    ;
      )     ;
      )     ;
      A     #Enable;
      =     #Ret_End_Aux;
NETWORK
TITLE =Ret End Program
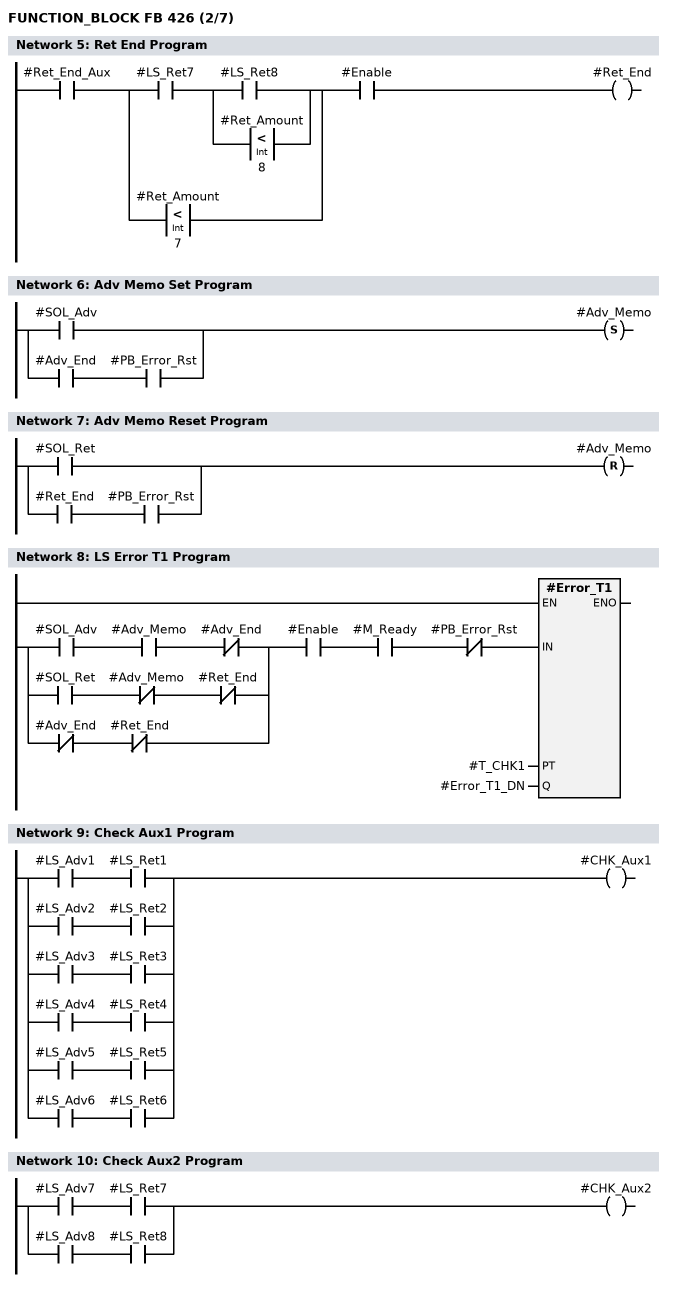

      A     #Ret_End_Aux;
      A(    ;
      A     #LS_Ret7;
      A(    ;
      O     #LS_Ret8;
      O(    ;
      L     #Ret_Amount;
      L     8;
      <I    ;
      )     ;
      )     ;
      O(    ;
      L     #Ret_Amount;
      L     7;
      <I    ;
      )     ;
      )     ;
      A     #Enable;
      =     #Ret_End;
NETWORK
TITLE =Adv Memo Set Program

      O     #SOL_Adv;
      O     ;
      A     #Adv_End;
      A     #PB_Error_Rst;
      S     #Adv_Memo;
NETWORK
TITLE =Adv Memo Reset Program

      O     #SOL_Ret;
      O     ;
      A     #Ret_End;
      A     #PB_Error_Rst;
      R     #Adv_Memo;
NETWORK
TITLE =LS Error T1 Program

      A(    ;
      A     #SOL_Adv;
      A     #Adv_Memo;
      AN    #Adv_End;
      O     ;
      A     #SOL_Ret;
      AN    #Adv_Memo;
      AN    #Ret_End;
      O     ;
      AN    #Adv_End;
      AN    #Ret_End;
      )     ;
      A     #Enable;
      A     #M_Ready;
      AN    #PB_Error_Rst;
      =     L      0.0;
      BLD   103;
      CALL #Error_T1 (
           IN                       := L      0.0,
           PT                       := #T_CHK1,
           Q                        := #Error_T1_DN);

      NOP   0;
NETWORK
TITLE =Check Aux1 Program

      A     #LS_Adv1;
      A     #LS_Ret1;
      O     ;
      A     #LS_Adv2;
      A     #LS_Ret2;
      O     ;
      A     #LS_Adv3;
      A     #LS_Ret3;
      O     ;
      A     #LS_Adv4;
      A     #LS_Ret4;
      O     ;
      A     #LS_Adv5;
      A     #LS_Ret5;
      O     ;
      A     #LS_Adv6;
      A     #LS_Ret6;
      =     #CHK_Aux1;
NETWORK
TITLE =Check Aux2 Program

      A     #LS_Adv7;
      A     #LS_Ret7;
      O     ;
      A     #LS_Adv8;
      A     #LS_Ret8;
      =     #CHK_Aux2;
NETWORK
TITLE =LS Error T2 Program
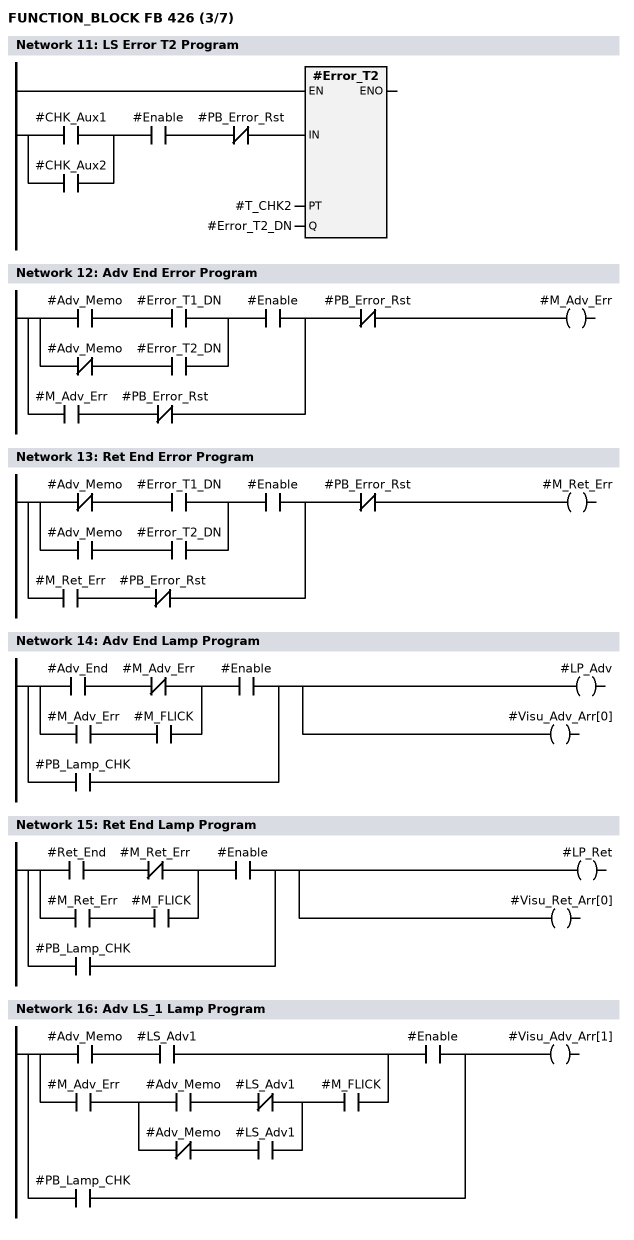

      A(    ;
      O     #CHK_Aux1;
      O     #CHK_Aux2;
      )     ;
      A     #Enable;
      AN    #PB_Error_Rst;
      =     L      0.0;
      BLD   103;
      CALL #Error_T2 (
           IN                       := L      0.0,
           PT                       := #T_CHK2,
           Q                        := #Error_T2_DN);

      NOP   0;
NETWORK
TITLE =Adv End Error Program

      A(    ;
      A(    ;
      A     #Adv_Memo;
      A     #Error_T1_DN;
      O     ;
      AN    #Adv_Memo;
      A     #Error_T2_DN;
      )     ;
      A     #Enable;
      O     ;
      A     #M_Adv_Err;
      AN    #PB_Error_Rst;
      )     ;
      AN    #PB_Error_Rst;
      =     #M_Adv_Err;
NETWORK
TITLE =Ret End Error Program

      A(    ;
      A(    ;
      AN    #Adv_Memo;
      A     #Error_T1_DN;
      O     ;
      A     #Adv_Memo;
      A     #Error_T2_DN;
      )     ;
      A     #Enable;
      O     ;
      A     #M_Ret_Err;
      AN    #PB_Error_Rst;
      )     ;
      AN    #PB_Error_Rst;
      =     #M_Ret_Err;
NETWORK
TITLE =Adv End Lamp Program

      A(    ;
      A     #Adv_End;
      AN    #M_Adv_Err;
      O     ;
      A     #M_Adv_Err;
      A     #M_FLICK;
      )     ;
      A     #Enable;
      O     #PB_Lamp_CHK;
      =     #LP_Adv;
      =     #Visu_Adv_Arr[0];
NETWORK
TITLE =Ret End Lamp Program

      A(    ;
      A     #Ret_End;
      AN    #M_Ret_Err;
      O     ;
      A     #M_Ret_Err;
      A     #M_FLICK;
      )     ;
      A     #Enable;
      O     #PB_Lamp_CHK;
      =     #LP_Ret;
      =     #Visu_Ret_Arr[0];
NETWORK
TITLE =Adv LS_1 Lamp Program

      A(    ;
      A     #Adv_Memo;
      A     #LS_Adv1;
      O     ;
      A     #M_Adv_Err;
      A(    ;
      A     #Adv_Memo;
      AN    #LS_Adv1;
      O     ;
      AN    #Adv_Memo;
      A     #LS_Adv1;
      )     ;
      A     #M_FLICK;
      )     ;
      A     #Enable;
      O     #PB_Lamp_CHK;
      =     #Visu_Adv_Arr[1];
NETWORK
TITLE =Adv LS_2 Lamp Program
//
//
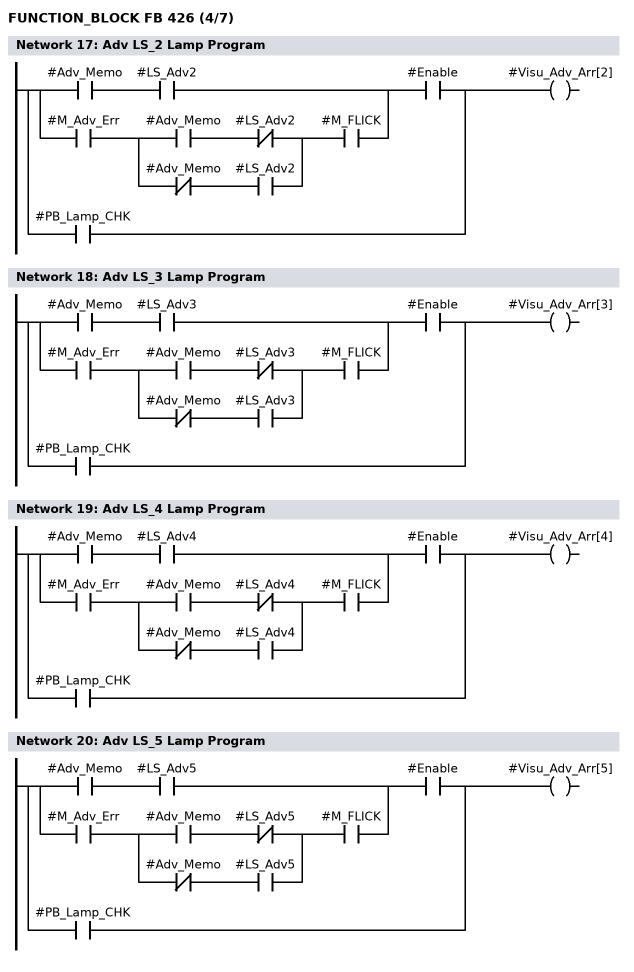
      A(    ;
      A     #Adv_Memo;
      A     #LS_Adv2;
      O     ;
      A     #M_Adv_Err;
      A(    ;
      A     #Adv_Memo;
      AN    #LS_Adv2;
      O     ;
      AN    #Adv_Memo;
      A     #LS_Adv2;
      )     ;
      A     #M_FLICK;
      )     ;
      A     #Enable;
      O     #PB_Lamp_CHK;
      =     #Visu_Adv_Arr[2];
NETWORK
TITLE =Adv LS_3 Lamp Program
//
//
      A(    ;
      A     #Adv_Memo;
      A     #LS_Adv3;
      O     ;
      A     #M_Adv_Err;
      A(    ;
      A     #Adv_Memo;
      AN    #LS_Adv3;
      O     ;
      AN    #Adv_Memo;
      A     #LS_Adv3;
      )     ;
      A     #M_FLICK;
      )     ;
      A     #Enable;
      O     #PB_Lamp_CHK;
      =     #Visu_Adv_Arr[3];
NETWORK
TITLE =Adv LS_4 Lamp Program
//
//
      A(    ;
      A     #Adv_Memo;
      A     #LS_Adv4;
      O     ;
      A     #M_Adv_Err;
      A(    ;
      A     #Adv_Memo;
      AN    #LS_Adv4;
      O     ;
      AN    #Adv_Memo;
      A     #LS_Adv4;
      )     ;
      A     #M_FLICK;
      )     ;
      A     #Enable;
      O     #PB_Lamp_CHK;
      =     #Visu_Adv_Arr[4];
NETWORK
TITLE =Adv LS_5 Lamp Program
//
//
      A(    ;
      A     #Adv_Memo;
      A     #LS_Adv5;
      O     ;
      A     #M_Adv_Err;
      A(    ;
      A     #Adv_Memo;
      AN    #LS_Adv5;
      O     ;
      AN    #Adv_Memo;
      A     #LS_Adv5;
      )     ;
      A     #M_FLICK;
      )     ;
      A     #Enable;
      O     #PB_Lamp_CHK;
      =     #Visu_Adv_Arr[5];
NETWORK
TITLE =Adv LS_6 Lamp Program
//
//
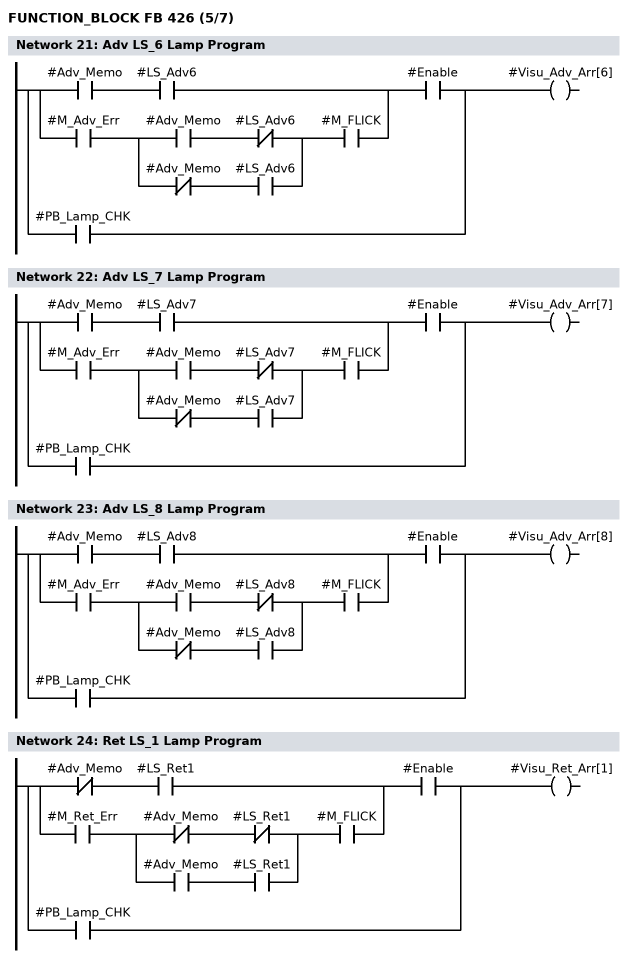
      A(    ;
      A     #Adv_Memo;
      A     #LS_Adv6;
      O     ;
      A     #M_Adv_Err;
      A(    ;
      A     #Adv_Memo;
      AN    #LS_Adv6;
      O     ;
      AN    #Adv_Memo;
      A     #LS_Adv6;
      )     ;
      A     #M_FLICK;
      )     ;
      A     #Enable;
      O     #PB_Lamp_CHK;
      =     #Visu_Adv_Arr[6];
NETWORK
TITLE =Adv LS_7 Lamp Program
//
//
      A(    ;
      A     #Adv_Memo;
      A     #LS_Adv7;
      O     ;
      A     #M_Adv_Err;
      A(    ;
      A     #Adv_Memo;
      AN    #LS_Adv7;
      O     ;
      AN    #Adv_Memo;
      A     #LS_Adv7;
      )     ;
      A     #M_FLICK;
      )     ;
      A     #Enable;
      O     #PB_Lamp_CHK;
      =     #Visu_Adv_Arr[7];
NETWORK
TITLE =Adv LS_8 Lamp Program
//
//
      A(    ;
      A     #Adv_Memo;
      A     #LS_Adv8;
      O     ;
      A     #M_Adv_Err;
      A(    ;
      A     #Adv_Memo;
      AN    #LS_Adv8;
      O     ;
      AN    #Adv_Memo;
      A     #LS_Adv8;
      )     ;
      A     #M_FLICK;
      )     ;
      A     #Enable;
      O     #PB_Lamp_CHK;
      =     #Visu_Adv_Arr[8];
NETWORK
TITLE =Ret LS_1 Lamp Program
//
//
      A(    ;
      AN    #Adv_Memo;
      A     #LS_Ret1;
      O     ;
      A     #M_Ret_Err;
      A(    ;
      AN    #Adv_Memo;
      AN    #LS_Ret1;
      O     ;
      A     #Adv_Memo;
      A     #LS_Ret1;
      )     ;
      A     #M_FLICK;
      )     ;
      A     #Enable;
      O     #PB_Lamp_CHK;
      =     #Visu_Ret_Arr[1];
NETWORK
TITLE =Ret LS_2 Lamp Program
//
//
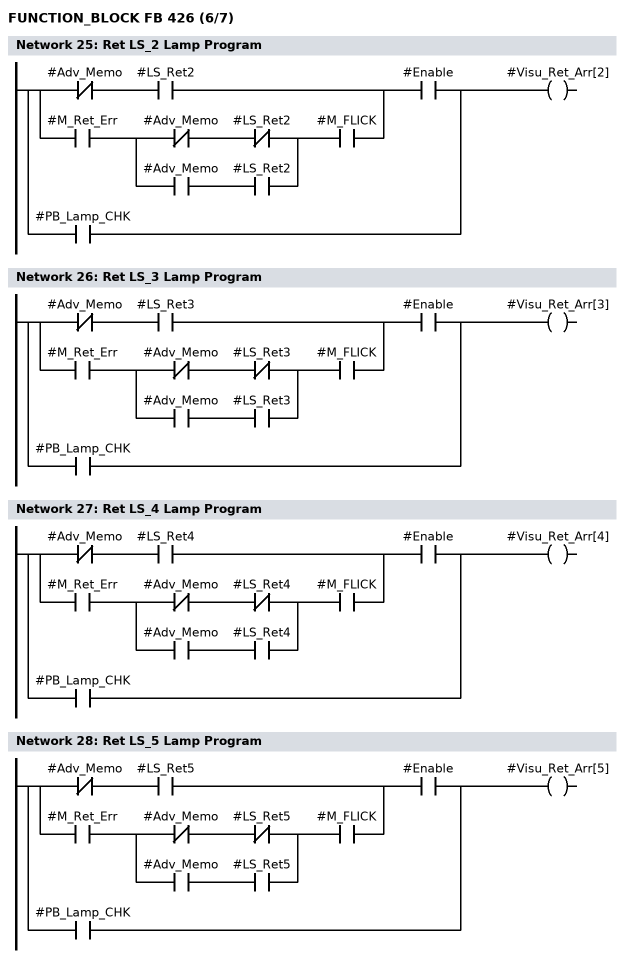
      A(    ;
      AN    #Adv_Memo;
      A     #LS_Ret2;
      O     ;
      A     #M_Ret_Err;
      A(    ;
      AN    #Adv_Memo;
      AN    #LS_Ret2;
      O     ;
      A     #Adv_Memo;
      A     #LS_Ret2;
      )     ;
      A     #M_FLICK;
      )     ;
      A     #Enable;
      O     #PB_Lamp_CHK;
      =     #Visu_Ret_Arr[2];
NETWORK
TITLE =Ret LS_3 Lamp Program
//
//
      A(    ;
      AN    #Adv_Memo;
      A     #LS_Ret3;
      O     ;
      A     #M_Ret_Err;
      A(    ;
      AN    #Adv_Memo;
      AN    #LS_Ret3;
      O     ;
      A     #Adv_Memo;
      A     #LS_Ret3;
      )     ;
      A     #M_FLICK;
      )     ;
      A     #Enable;
      O     #PB_Lamp_CHK;
      =     #Visu_Ret_Arr[3];
NETWORK
TITLE =Ret LS_4 Lamp Program
//
//
      A(    ;
      AN    #Adv_Memo;
      A     #LS_Ret4;
      O     ;
      A     #M_Ret_Err;
      A(    ;
      AN    #Adv_Memo;
      AN    #LS_Ret4;
      O     ;
      A     #Adv_Memo;
      A     #LS_Ret4;
      )     ;
      A     #M_FLICK;
      )     ;
      A     #Enable;
      O     #PB_Lamp_CHK;
      =     #Visu_Ret_Arr[4];
NETWORK
TITLE =Ret LS_5 Lamp Program
//
//
      A(    ;
      AN    #Adv_Memo;
      A     #LS_Ret5;
      O     ;
      A     #M_Ret_Err;
      A(    ;
      AN    #Adv_Memo;
      AN    #LS_Ret5;
      O     ;
      A     #Adv_Memo;
      A     #LS_Ret5;
      )     ;
      A     #M_FLICK;
      )     ;
      A     #Enable;
      O     #PB_Lamp_CHK;
      =     #Visu_Ret_Arr[5];
NETWORK
TITLE =Ret LS_6 Lamp Program
//
//
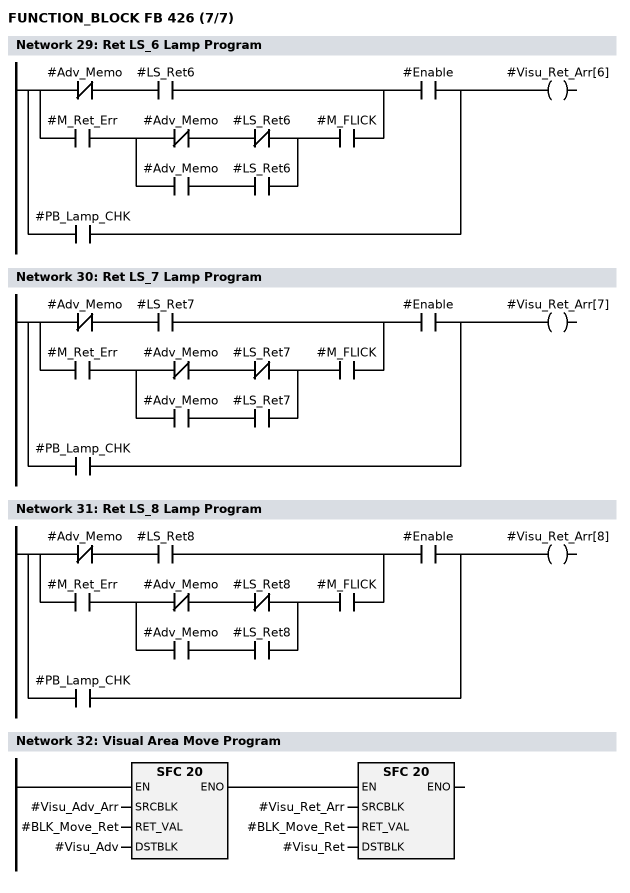
      A(    ;
      AN    #Adv_Memo;
      A     #LS_Ret6;
      O     ;
      A     #M_Ret_Err;
      A(    ;
      AN    #Adv_Memo;
      AN    #LS_Ret6;
      O     ;
      A     #Adv_Memo;
      A     #LS_Ret6;
      )     ;
      A     #M_FLICK;
      )     ;
      A     #Enable;
      O     #PB_Lamp_CHK;
      =     #Visu_Ret_Arr[6];
NETWORK
TITLE =Ret LS_7 Lamp Program
//
//
      A(    ;
      AN    #Adv_Memo;
      A     #LS_Ret7;
      O     ;
      A     #M_Ret_Err;
      A(    ;
      AN    #Adv_Memo;
      AN    #LS_Ret7;
      O     ;
      A     #Adv_Memo;
      A     #LS_Ret7;
      )     ;
      A     #M_FLICK;
      )     ;
      A     #Enable;
      O     #PB_Lamp_CHK;
      =     #Visu_Ret_Arr[7];
NETWORK
TITLE =Ret LS_8 Lamp Program
//
//
      A(    ;
      AN    #Adv_Memo;
      A     #LS_Ret8;
      O     ;
      A     #M_Ret_Err;
      A(    ;
      AN    #Adv_Memo;
      AN    #LS_Ret8;
      O     ;
      A     #Adv_Memo;
      A     #LS_Ret8;
      )     ;
      A     #M_FLICK;
      )     ;
      A     #Enable;
      O     #PB_Lamp_CHK;
      =     #Visu_Ret_Arr[8];
NETWORK
TITLE =Visual Area Move Program

      A(    ;
      CALL SFC   20 (
           SRCBLK                   := #Visu_Adv_Arr,
           RET_VAL                  := #BLK_Move_Ret,
           DSTBLK                   := #Visu_Adv);
      A     BR;
      )     ;
      JNB   _001;
      CALL SFC   20 (
           SRCBLK                   := #Visu_Ret_Arr,
           RET_VAL                  := #BLK_Move_Ret,
           DSTBLK                   := #Visu_Ret);
_001: NOP   0;
END_FUNCTION_BLOCK

FUNCTION_BLOCK FB 470
TITLE =HMI Body Type Modify Variables Program
AUTHOR : HMC
FAMILY : HMI
NAME : HMI
VERSION : 1.0


VAR_INPUT
  Station : INT ;
  HMI_Disp_DB : INT ;
  HMI_Disp_Add : INT ;
  CType_DB : INT ;
  CType_Start_Add : INT ;
  Byte_per_Stn : INT ;
  M_Modify_OK : BOOL ;
  SS_CCR_On : BOOL ;
  PB_Set : BOOL ;
  PB_Reset : BOOL ;
END_VAR
VAR_OUTPUT
  LP_CCR_On : BOOL ;
  LP_Modify_On : BOOL ;
END_VAR
VAR
  Source_Data : WORD ;
  Modify_Data : WORD ;
  Pre_Station : INT ;
  Station_PLS : BOOL ;
  Source_Add : INT ;
  SFC20_Ret : INT ;
  Fill_Source : WORD ;
END_VAR
VAR_TEMP
  Source_Area : ANY ;
  Modify_Area : ANY ;
END_VAR
BEGIN
NETWORK
TITLE =FAC On Lamp Program

      A     #SS_CCR_On;
      =     #LP_CCR_On;
NETWORK
TITLE =Operation Pulse

      L     #Station; // Station Select Data
      L     0; // Is Not Zero
      <>I   ;
      JNB   _End; // Jump to End
NETWORK
TITLE =Modify On Lamp Program
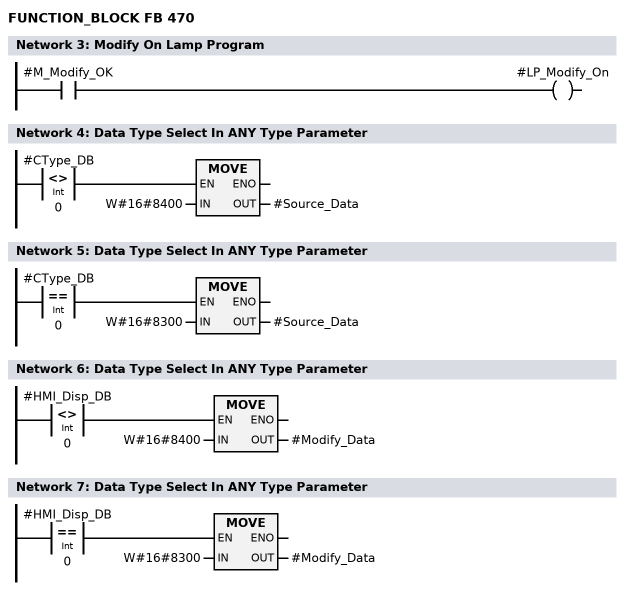

      A     #M_Modify_OK;
      =     #LP_Modify_On;
NETWORK
TITLE =Data Type Select In ANY Type Parameter

      A(    ; // If Source DB is Not Zero
      L     #CType_DB;
      L     0;
      <>I   ;
      )     ;
      JNB   _B01; // Jump to Next Step
      L     W#16#8400; // Load "8400" _ Means "DB Area"
      T     #Source_Data; // Transfer to Data_Type
_B01: NOP   0;
NETWORK
TITLE =Data Type Select In ANY Type Parameter

      A(    ; // If DB_NO is Zero
      L     #CType_DB;
      L     0;
      ==I   ;
      )     ;
      JNB   _B02; // Jump to Next Step
      L     W#16#8300; // Load "8300" _ Means "Bit Memory Area"
      T     #Source_Data; // Transfer to Data_Type
_B02: NOP   0;
NETWORK
TITLE =Data Type Select In ANY Type Parameter

      A(    ; // If Source DB is Not Zero
      L     #HMI_Disp_DB;
      L     0;
      <>I   ;
      )     ;
      JNB   _B03; // Jump to Next Step
      L     W#16#8400; // Load "8400" _ Means "DB Area"
      T     #Modify_Data; // Transfer to Data_Type
_B03: NOP   0;
NETWORK
TITLE =Data Type Select In ANY Type Parameter

      A(    ; // If DB_NO is Zero
      L     #HMI_Disp_DB;
      L     0;
      ==I   ;
      )     ;
      JNB   _B04; // Jump to Next Step
      L     W#16#8300; // Load "8300" _ Means "Bit Memory Area"
      T     #Modify_Data; // Transfer to Data_Type
_B04: NOP   0;
NETWORK
TITLE =Source Area Start Address Calculate Porgram

      L     #Station; // Station Amount - 1
      L     1;
      -I    ;
      L     #Byte_per_Stn; // Multi Length Per Station
      *I    ;
      L     #CType_Start_Add;
      +I    ;
      T     #Source_Add;
NETWORK
TITLE =Make a "ANY" Type Data

      LAR1  P##Source_Area; // Load 1st Station Address of ANY Pointer In "AR1"

      L     B#16#10; // Load Syntax ID For S7 "10"
      T     LB [AR1,P#0.0]; // Transfer ID to the ANY Pointer

      L     B#16#2; // Load Data Type _ "2" means "BYTE"
      T     LB [AR1,P#1.0]; // Transfer Data Type to the ANY Pointer

      L     #Byte_per_Stn; // Load the Length of Source Data
      T     LW [AR1,P#2.0]; // Transfer the Numbers to the ANY Pointer

      L     #CType_DB; // Load DB Number _ "0" means don't use "DB"
      T     LW [AR1,P#4.0]; // Transfer the Numbers to the ANY Pointer

      L     #Source_Data; // Load Data Type _ "83" means "Bit Memory" Area
      T     LW [AR1,P#6.0]; //                  "84" means "DB" Area

      L     #Source_Add; // Load Start Address
      SLW   3; // Shift Left Word _ "3" Bit
      T     LW [AR1,P#8.0]; // Transfer the Address to the ANY Pointer

      LAR1  P##Modify_Area; // Load 2nd Station Address of ANY Pointer In "AR1"

      L     B#16#10; //Load Syntax ID For S7 "10"
      T     LB [AR1,P#0.0]; //Load Syntax ID For S7 "10"

      L     B#16#2; //  Load Data Type _ "2" means "BYTE"
      T     LB [AR1,P#1.0]; // Transfer Data Type to the ANY Pointer

      L     #Byte_per_Stn; // Load the Length of Target Data
      T     LW [AR1,P#2.0]; // Transfer the Numbers to the ANY Pointer

      L     #HMI_Disp_DB; // Load DB Number _ "0" means don't use "DB"
      T     LW [AR1,P#4.0]; // Transfer the Numbers to the ANY Pointer

      L     #Modify_Data; // Load Data Type _ "83" means "Bit Memory" Area
      T     LW [AR1,P#6.0]; //                  "84" means "DB" Area

      L     #HMI_Disp_Add; //  Load Start Address
      SLW   3; // Shift Left Word _ "3" Bit
      T     LW [AR1,P#8.0]; // Transfer the Address to the ANY Pointer

NETWORK
TITLE =Copy To Modify Area Program

      L     #Station;
      L     #Pre_Station;
      <>I   ;
      JNB   _B05;
NETWORK
TITLE =Copy To Previous Station No Program

      L     #Station;
      T     #Pre_Station;
NETWORK
TITLE =Block Move to Modify Area


      CALL SFC   20 (
           SRCBLK                   := #Source_Area,
           RET_VAL                  := #SFC20_Ret,
           DSTBLK                   := #Modify_Area);
_B05: NOP   0;
NETWORK
TITLE =Data Clear Program

      A     #M_Modify_OK;
      A     #PB_Reset;
      JNB   _B06;
NETWORK
TITLE =Clear Source Data Area


      CALL SFC   21 (
           IN0                      := #Fill_Source,// "Zero"
           RET_VAL                  := #SFC20_Ret,
           OUT1                     := #Source_Area);// Transfer to First Station Area

NETWORK
TITLE =Clear Source Data Area


      CALL SFC   21 (
           IN0                      := #Fill_Source,// "Zero"
           RET_VAL                  := #SFC20_Ret,
           OUT1                     := #Modify_Area);// Transfer to First Station Area
_B06: NOP   0;
NETWORK
TITLE =Data Clear Program

      A     #M_Modify_OK;
      A     #PB_Set;
      JNB   _B07;
NETWORK
TITLE =Block Move to Modify Area


      CALL SFC   20 (
           SRCBLK                   := #Modify_Area,
           RET_VAL                  := #SFC20_Ret,
           DSTBLK                   := #Source_Area);
_B07: NOP   0;
NETWORK
TITLE =


_End: NOP   0;

END_FUNCTION_BLOCK

FUNCTION_BLOCK FB 475
TITLE =ProfiBus DP Communication Fault Variables Program
AUTHOR : HMC
FAMILY : Drive
NAME : Drive
VERSION : 1.0


VAR_INPUT
  M_Check_Active : BOOL ;
  DP_Not_Pre_Byte : BYTE ;	//Startadress Outputs from HW-Konfig
  DP_Error_Byte : BYTE ;	//Startadress Inputs from HW-Konfig
  M_Error_Rst : BOOL ;
END_VAR
VAR_OUTPUT
  Node0_Fault : BOOL ;
  Node1_Fault : BOOL ;
  Node2_Fault : BOOL ;
  Node3_Fault : BOOL ;
  Node4_Fault : BOOL ;
  Node5_Fault : BOOL ;
  Node6_Fault : BOOL ;
  Node7_Fault : BOOL ;
END_VAR
VAR
  Pre_Arr : ARRAY  [0 .. 7 ] OF BOOL ;
  Fault_Arr : ARRAY  [0 .. 7 ] OF BOOL ;
  node_0_err : SFB 4;
  node_1_err : SFB 4;
  node_2_err : SFB 4;
  node_3_err : SFB 4;
  node_4_err : SFB 4;
  node_5_err : SFB 4;
  node_6_err : SFB 4;
  node_7_err : SFB 4;
END_VAR
VAR_TEMP
  Ret : INT ;
END_VAR
BEGIN
NETWORK
TITLE =DP Fault Byte Move To DP Fault Array
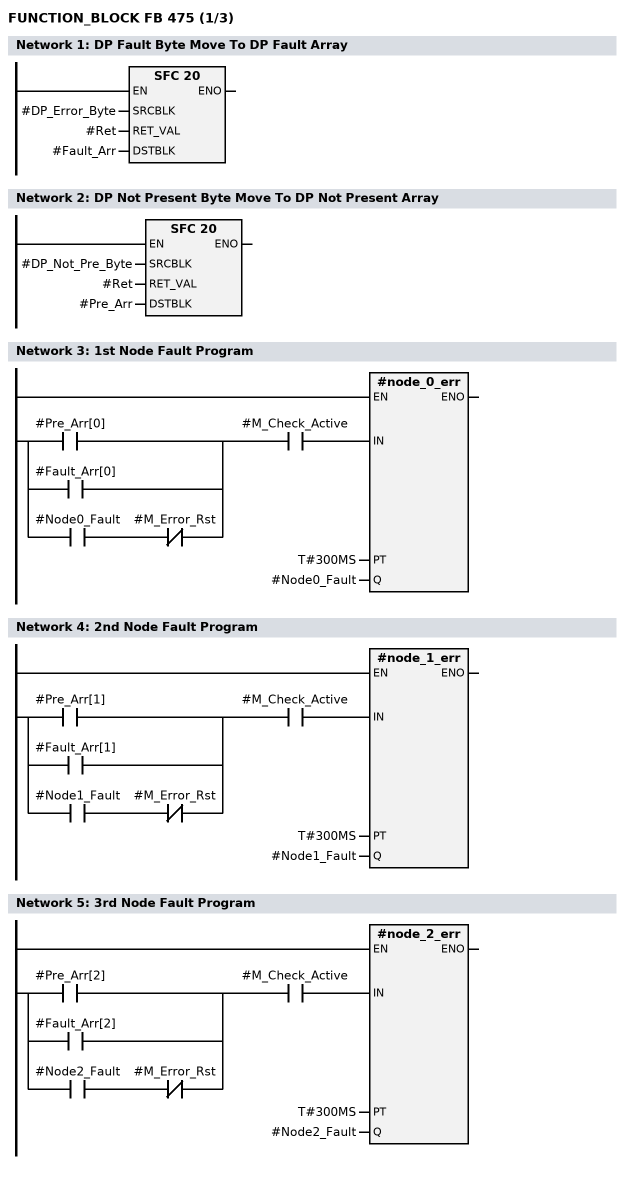

      CALL SFC   20 (
           SRCBLK                   := #DP_Error_Byte,
           RET_VAL                  := #Ret,
           DSTBLK                   := #Fault_Arr);
      NOP   0;
NETWORK
TITLE =DP Not Present Byte Move To DP Not Present Array

      CALL SFC   20 (
           SRCBLK                   := #DP_Not_Pre_Byte,
           RET_VAL                  := #Ret,
           DSTBLK                   := #Pre_Arr);
      NOP   0;
NETWORK
TITLE =1st Node Fault Program

      A(    ;
      O     #Pre_Arr[0];
      O     #Fault_Arr[0];
      O     ;
      A     #Node0_Fault;
      AN    #M_Error_Rst;
      )     ;
      A     #M_Check_Active;
      =     L      2.0;
      BLD   103;
      CALL #node_0_err (
           IN                       := L      2.0,
           PT                       := T#300MS,
           Q                        := #Node0_Fault);

      NOP   0;
NETWORK
TITLE =2nd Node Fault Program

      A(    ;
      O     #Pre_Arr[1];
      O     #Fault_Arr[1];
      O     ;
      A     #Node1_Fault;
      AN    #M_Error_Rst;
      )     ;
      A     #M_Check_Active;
      =     L      2.0;
      BLD   103;
      CALL #node_1_err (
           IN                       := L      2.0,
           PT                       := T#300MS,
           Q                        := #Node1_Fault);

      NOP   0;
NETWORK
TITLE =3rd Node Fault Program

      A(    ;
      O     #Pre_Arr[2];
      O     #Fault_Arr[2];
      O     ;
      A     #Node2_Fault;
      AN    #M_Error_Rst;
      )     ;
      A     #M_Check_Active;
      =     L      2.0;
      BLD   103;
      CALL #node_2_err (
           IN                       := L      2.0,
           PT                       := T#300MS,
           Q                        := #Node2_Fault);

      NOP   0;
NETWORK
TITLE =4th Node Fault Program
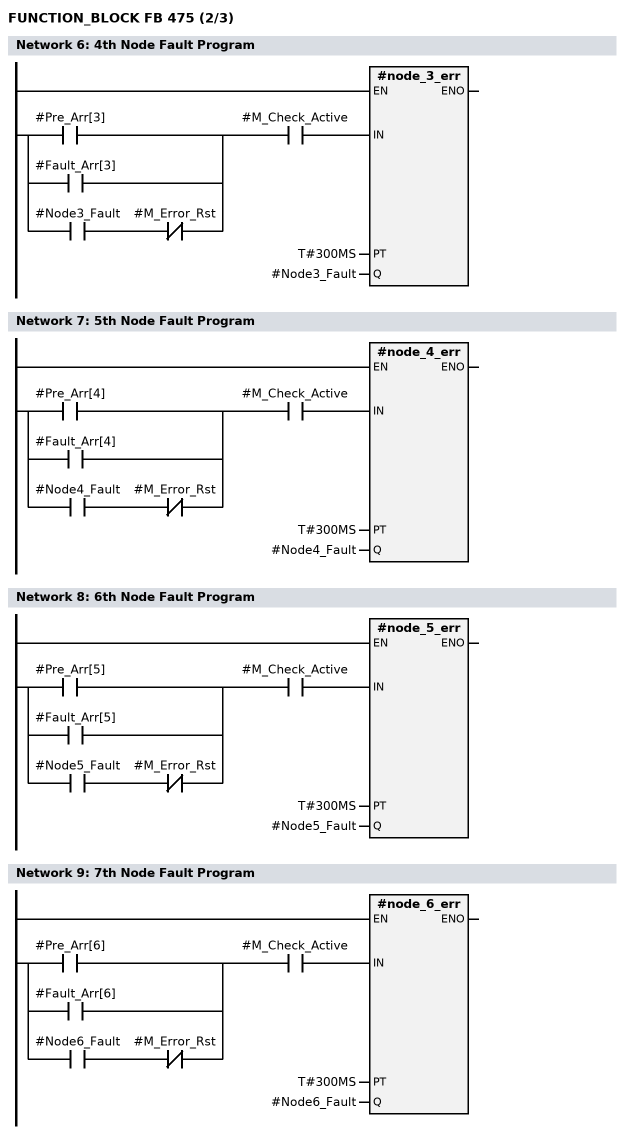

      A(    ;
      O     #Pre_Arr[3];
      O     #Fault_Arr[3];
      O     ;
      A     #Node3_Fault;
      AN    #M_Error_Rst;
      )     ;
      A     #M_Check_Active;
      =     L      2.0;
      BLD   103;
      CALL #node_3_err (
           IN                       := L      2.0,
           PT                       := T#300MS,
           Q                        := #Node3_Fault);

      NOP   0;
NETWORK
TITLE =5th Node Fault Program

      A(    ;
      O     #Pre_Arr[4];
      O     #Fault_Arr[4];
      O     ;
      A     #Node4_Fault;
      AN    #M_Error_Rst;
      )     ;
      A     #M_Check_Active;
      =     L      2.0;
      BLD   103;
      CALL #node_4_err (
           IN                       := L      2.0,
           PT                       := T#300MS,
           Q                        := #Node4_Fault);

      NOP   0;
NETWORK
TITLE =6th Node Fault Program

      A(    ;
      O     #Pre_Arr[5];
      O     #Fault_Arr[5];
      O     ;
      A     #Node5_Fault;
      AN    #M_Error_Rst;
      )     ;
      A     #M_Check_Active;
      =     L      2.0;
      BLD   103;
      CALL #node_5_err (
           IN                       := L      2.0,
           PT                       := T#300MS,
           Q                        := #Node5_Fault);

      NOP   0;
NETWORK
TITLE =7th Node Fault Program

      A(    ;
      O     #Pre_Arr[6];
      O     #Fault_Arr[6];
      O     ;
      A     #Node6_Fault;
      AN    #M_Error_Rst;
      )     ;
      A     #M_Check_Active;
      =     L      2.0;
      BLD   103;
      CALL #node_6_err (
           IN                       := L      2.0,
           PT                       := T#300MS,
           Q                        := #Node6_Fault);

      NOP   0;
NETWORK
TITLE =8th Node Fault Program
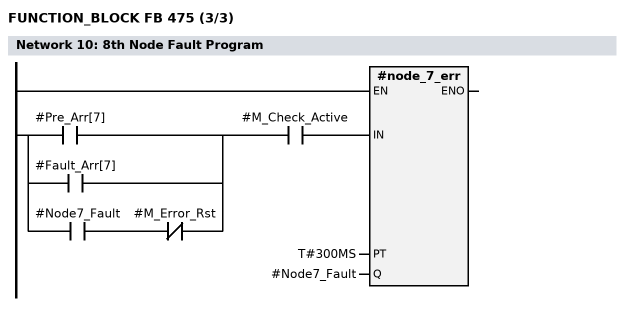

      A(    ;
      O     #Pre_Arr[7];
      O     #Fault_Arr[7];
      O     ;
      A     #Node7_Fault;
      AN    #M_Error_Rst;
      )     ;
      A     #M_Check_Active;
      =     L      2.0;
      BLD   103;
      CALL #node_7_err (
           IN                       := L      2.0,
           PT                       := T#300MS,
           Q                        := #Node7_Fault);

      NOP   0;
END_FUNCTION_BLOCK

FUNCTION_BLOCK FB 512
TITLE =Car Type Variables Program
AUTHOR : HMC
FAMILY : Car_Type
NAME : Car_Type
VERSION : 1.0


VAR_INPUT
  Stn_Vin_No : DINT ;	//Startadress Inputs from HW-Konfig
  Stn_Bt_1Word : WORD ;
  Stn_Bt_2Word : WORD ;
  Stn_Bt_3Word : WORD ;
  Stn_Bt_4Word : WORD ;
  Stn_Bt_5Word_Sp : WORD ;
  Stn_Bt_6Word_Sp : WORD ;
END_VAR
VAR_OUTPUT
  M_BType_On : BOOL ;
  M_BType_None : BOOL ;
  M_Bypass_BType : BOOL ;
  M_BType_TL : BOOL ;
  M_BType_LM : BOOL ;
  M_BType_SP1 : BOOL ;
  M_BType_SP2 : BOOL ;
  M_BType_SP3 : BOOL ;
  M_BType_DOM : BOOL ;
  M_BType_EXP : BOOL ;
  Robot_Prog_No : INT ;
END_VAR
VAR
  STN_Btype_1Arr : ARRAY  [0 .. 15 ] OF BOOL ;
  STN_Btype_2Arr : ARRAY  [0 .. 15 ] OF BOOL ;
  STN_Btype_3Arr : ARRAY  [0 .. 15 ] OF BOOL ;
  STN_Btype_4Arr : ARRAY  [0 .. 15 ] OF BOOL ;
  STN_Btype_5Arr : ARRAY  [0 .. 15 ] OF BOOL ;
  STN_Btype_6Arr : ARRAY  [0 .. 15 ] OF BOOL ;
  STN_1st_BT_On : BOOL ;
  STN_2nd_BT_On : BOOL ;
  STN_3rd_BT_On : BOOL ;
  STN_4th_BT_On : BOOL ;
  STN_5th_BT_On : BOOL ;
  STN_6th_BT_On : BOOL ;
  STN_7th_BT_On : BOOL ;
  STN_8th_BT_On : BOOL ;
  STN_9th_BT_On : BOOL ;
  STN_10th_BT_On : BOOL ;
  STN_11th_BT_On : BOOL ;
  STN_12th_BT_On : BOOL ;
  STN_1st_BT_Off : BOOL ;
  BLKMove_Ret : INT ;
  VIN_1BCD : WORD ;
  VIN_2BCD : WORD ;
  VIN_1Int : INT ;
  VIN_2Int : INT ;
END_VAR
BEGIN
NETWORK
TITLE =Station Body Type Data Change to 16-bit array

      CALL SFC   20 (
           SRCBLK                   := #Stn_Bt_1Word,
           RET_VAL                  := #BLKMove_Ret,
           DSTBLK                   := #STN_Btype_1Arr);
      NOP   0;
NETWORK
TITLE =Station Body Type Data Change to 16-bit array

      CALL SFC   20 (
           SRCBLK                   := #Stn_Bt_2Word,
           RET_VAL                  := #BLKMove_Ret,
           DSTBLK                   := #STN_Btype_2Arr);
      NOP   0;
NETWORK
TITLE =Station Body Type Data Change to 16-bit array

      CALL SFC   20 (
           SRCBLK                   := #Stn_Bt_3Word,
           RET_VAL                  := #BLKMove_Ret,
           DSTBLK                   := #STN_Btype_3Arr);
      NOP   0;
NETWORK
TITLE =Station Body Type Data Change to 16-bit array

      CALL SFC   20 (
           SRCBLK                   := #Stn_Bt_4Word,
           RET_VAL                  := #BLKMove_Ret,
           DSTBLK                   := #STN_Btype_4Arr);
      NOP   0;
NETWORK
TITLE =Station Body Type Data Change to 16-bit array

      CALL SFC   20 (
           SRCBLK                   := #Stn_Bt_5Word_Sp,
           RET_VAL                  := #BLKMove_Ret,
           DSTBLK                   := #STN_Btype_5Arr);
      NOP   0;
NETWORK
TITLE =Station Body Type Data Change to 16-bit array

      CALL SFC   20 (
           SRCBLK                   := #Stn_Bt_6Word_Sp,
           RET_VAL                  := #BLKMove_Ret,
           DSTBLK                   := #STN_Btype_6Arr);
      NOP   0;
NETWORK
TITLE =공정 1차종

      AN    OV;
      A(    ;
      O     #STN_Btype_1Arr[0];
      O     #STN_Btype_1Arr[1];
      O     #STN_Btype_1Arr[2];
      O     #STN_Btype_1Arr[3];
      O     #STN_Btype_1Arr[4];
      )     ;
      =     #STN_1st_BT_On;
NETWORK
TITLE =공정 2차종

      AN    OV;
      A(    ;
      O     #STN_Btype_1Arr[5];
      O     #STN_Btype_1Arr[6];
      O     #STN_Btype_1Arr[7];
      O     #STN_Btype_1Arr[8];
      )     ;
      =     #STN_2nd_BT_On;
NETWORK
TITLE =공정 3차종

      AN    OV;
      A(    ;
      O     #STN_Btype_1Arr[9];
      O     #STN_Btype_1Arr[10];
      )     ;
      =     #STN_3rd_BT_On;
NETWORK
TITLE =공정 4차종

      AN    OV;
      A(    ;
      O     #STN_Btype_1Arr[11];
      O     #STN_Btype_1Arr[12];
      O     #STN_Btype_1Arr[13];
      O     #STN_Btype_1Arr[14];
      O     #STN_Btype_1Arr[15];
      O     #STN_Btype_2Arr[0];
      O     #STN_Btype_2Arr[1];
      O     #STN_Btype_2Arr[2];
      O     #STN_Btype_2Arr[3];
      O     #STN_Btype_2Arr[4];
      O     #STN_Btype_2Arr[5];
      )     ;
      =     #STN_4th_BT_On;
NETWORK
TITLE =공정 5차종

      AN    OV;
      A(    ;
      O     #STN_Btype_2Arr[6];
      O     #STN_Btype_2Arr[7];
      )     ;
      =     #STN_5th_BT_On;
NETWORK
TITLE =공정 6차종

      AN    OV;
      A(    ;
      O     #STN_Btype_2Arr[8];
      O     #STN_Btype_2Arr[9];
      O     #STN_Btype_2Arr[10];
      O     #STN_Btype_2Arr[11];
      O     #STN_Btype_2Arr[12];
      O     #STN_Btype_2Arr[13];
      O     #STN_Btype_2Arr[14];
      O     #STN_Btype_2Arr[15];
      )     ;
      =     #STN_6th_BT_On;
NETWORK
TITLE =공정 7차종

      AN    OV;
      A(    ;
      O     #STN_Btype_3Arr[0];
      O     #STN_Btype_3Arr[1];
      )     ;
      =     #STN_7th_BT_On;
NETWORK
TITLE =공정 8차종

      AN    OV;
      A(    ;
      O     #STN_Btype_3Arr[2];
      O     #STN_Btype_3Arr[3];
      O     #STN_Btype_3Arr[6];
      )     ;
      =     #STN_8th_BT_On;
NETWORK
TITLE =공정 9차종

      AN    OV;
      A(    ;
      O     #STN_Btype_3Arr[4];
      O     #STN_Btype_3Arr[5];
      )     ;
      =     #STN_9th_BT_On;
NETWORK
TITLE =공정 10차종

      AN    OV;
      A(    ;
      O     #STN_Btype_3Arr[6];
      O     #STN_Btype_3Arr[7];
      ON    #STN_10th_BT_On;
      )     ;
      =     #STN_10th_BT_On;
NETWORK
TITLE =공정 11차종

      AN    OV;
      A(    ;
      O     #STN_Btype_3Arr[8];
      O     #STN_Btype_3Arr[9];
      O     #STN_Btype_3Arr[10];
      O     #STN_Btype_3Arr[11];
      O     #STN_Btype_3Arr[12];
      O     #STN_Btype_3Arr[13];
      O     #STN_Btype_3Arr[14];
      O     #STN_Btype_3Arr[15];
      O     #STN_Btype_4Arr[0];
      O     #STN_Btype_4Arr[1];
      O     #STN_Btype_4Arr[2];
      O     #STN_Btype_4Arr[3];
      O     #STN_Btype_4Arr[4];
      O     #STN_Btype_4Arr[5];
      O     #STN_Btype_4Arr[6];
      O     #STN_Btype_4Arr[7];
      O     #STN_Btype_4Arr[8];
      O     #STN_Btype_4Arr[9];
      )     ;
      =     #STN_11th_BT_On;
NETWORK
TITLE =공정 차종 있음
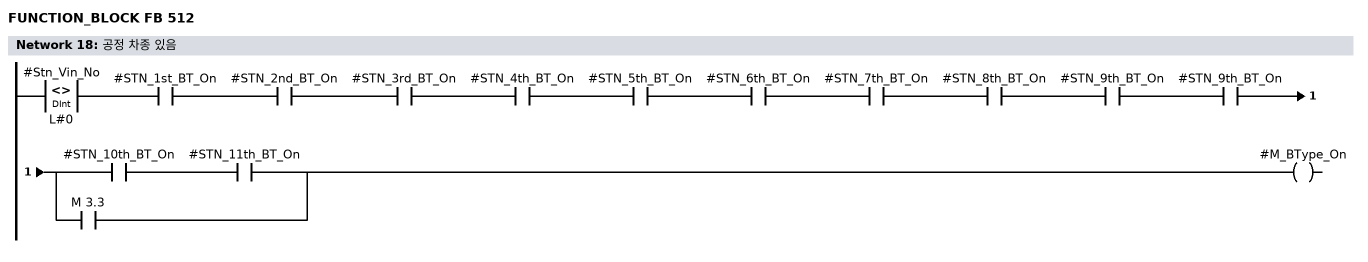

      A(    ;
      L     #Stn_Vin_No;
      L     L#0;
      <>D   ;
      )     ;
      A     #STN_1st_BT_On;
      A     #STN_2nd_BT_On;
      A     #STN_3rd_BT_On;
      A     #STN_4th_BT_On;
      A     #STN_5th_BT_On;
      A     #STN_6th_BT_On;
      A     #STN_7th_BT_On;
      A     #STN_8th_BT_On;
      A     #STN_9th_BT_On;
      A     #STN_9th_BT_On;
      A(    ;
      A     #STN_10th_BT_On;
      A     #STN_11th_BT_On;
      O     M      3.3;
      )     ;
      =     #M_BType_On;
NETWORK
TITLE =1차종 없음

      AN    OV;
      AN    #STN_Btype_1Arr[0];
      AN    #STN_Btype_1Arr[1];
      AN    #STN_Btype_1Arr[2];
      AN    #STN_Btype_1Arr[3];
      AN    #STN_Btype_1Arr[4];
      =     #STN_1st_BT_Off;
NETWORK
TITLE =공정 차종 없음
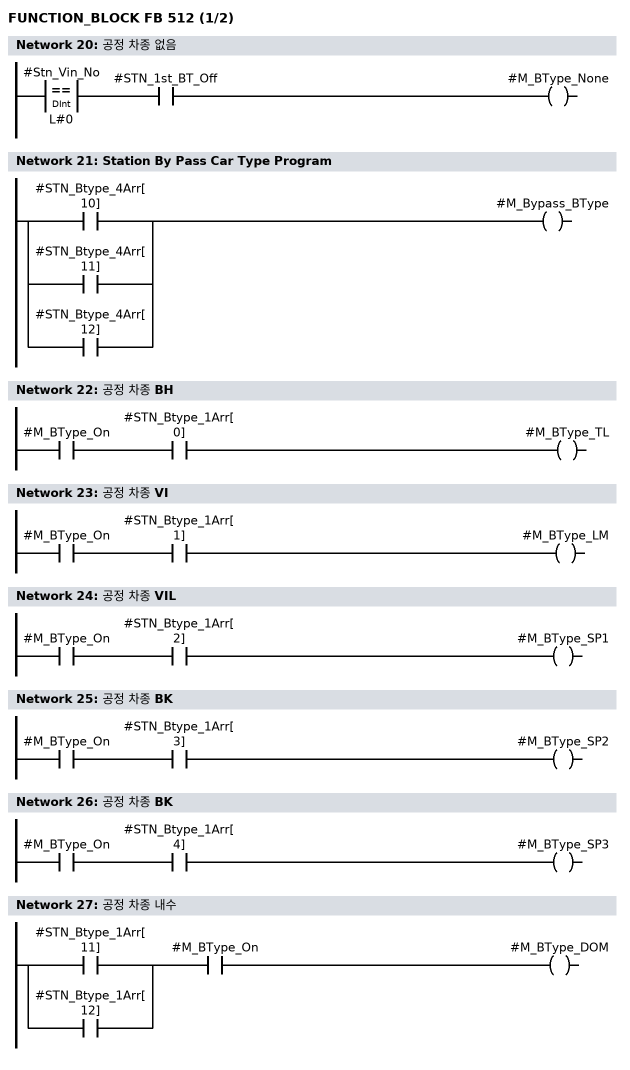

      A(    ;
      L     #Stn_Vin_No;
      L     L#0;
      ==D   ;
      )     ;
      A     #STN_1st_BT_Off;
      =     #M_BType_None;
NETWORK
TITLE =Station By Pass Car Type Program

      O     #STN_Btype_4Arr[10];
      O     #STN_Btype_4Arr[11];
      O     #STN_Btype_4Arr[12];
      =     #M_Bypass_BType;
NETWORK
TITLE =공정 차종 BH

      A     #M_BType_On;
      A     #STN_Btype_1Arr[0];
      =     #M_BType_TL;
NETWORK
TITLE =공정 차종 VI

      A     #M_BType_On;
      A     #STN_Btype_1Arr[1];
      =     #M_BType_LM;
NETWORK
TITLE =공정 차종 VIL

      A     #M_BType_On;
      A     #STN_Btype_1Arr[2];
      =     #M_BType_SP1;
NETWORK
TITLE =공정 차종 BK

      A     #M_BType_On;
      A     #STN_Btype_1Arr[3];
      =     #M_BType_SP2;
NETWORK
TITLE =공정 차종 BK

      A     #M_BType_On;
      A     #STN_Btype_1Arr[4];
      =     #M_BType_SP3;
NETWORK
TITLE =공정 차종 내수

      A(    ;
      O     #STN_Btype_1Arr[11];
      O     #STN_Btype_1Arr[12];
      )     ;
      A     #M_BType_On;
      =     #M_BType_DOM;
NETWORK
TITLE =공정 차종 수출
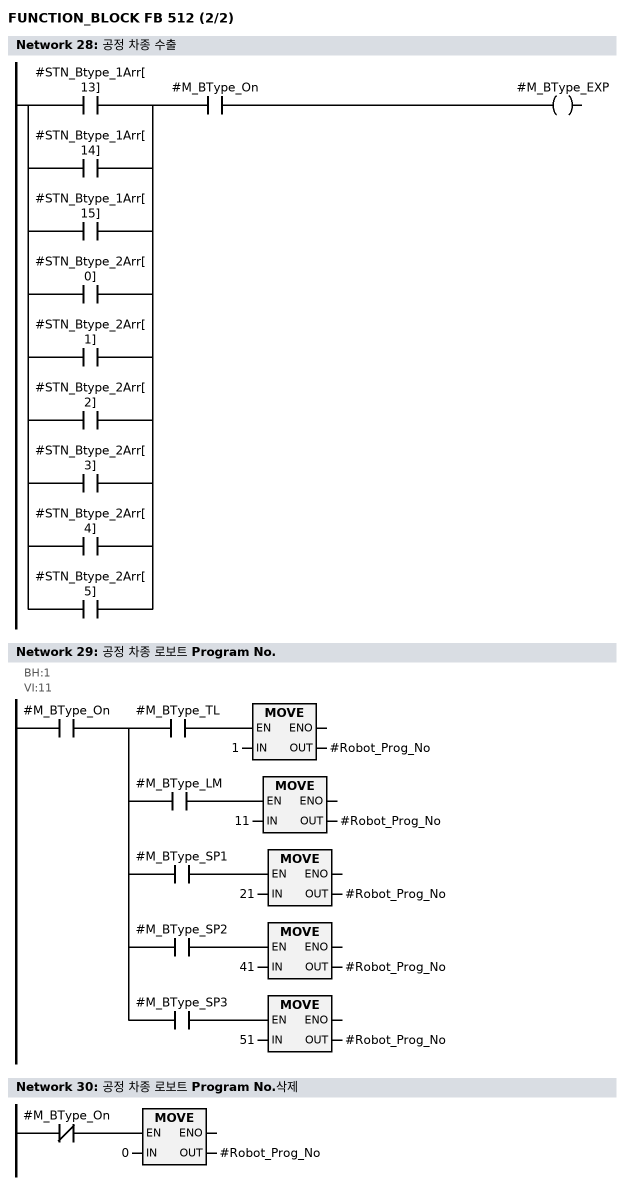

      A(    ;
      O     #STN_Btype_1Arr[13];
      O     #STN_Btype_1Arr[14];
      O     #STN_Btype_1Arr[15];
      O     #STN_Btype_2Arr[0];
      O     #STN_Btype_2Arr[1];
      O     #STN_Btype_2Arr[2];
      O     #STN_Btype_2Arr[3];
      O     #STN_Btype_2Arr[4];
      O     #STN_Btype_2Arr[5];
      )     ;
      A     #M_BType_On;
      =     #M_BType_EXP;
NETWORK
TITLE =공정 차종 로보트 Program No.
//BH:1
//VI:11
      A     #M_BType_On;
      =     L      0.0;
      A     L      0.0;
      A     #M_BType_TL;
      JNB   _001;
      L     1;
      T     #Robot_Prog_No;
_001: NOP   0;
      A     L      0.0;
      A     #M_BType_LM;
      JNB   _002;
      L     11;
      T     #Robot_Prog_No;
_002: NOP   0;
      A     L      0.0;
      A     #M_BType_SP1;
      JNB   _003;
      L     21;
      T     #Robot_Prog_No;
_003: NOP   0;
      A     L      0.0;
      A     #M_BType_SP2;
      JNB   _004;
      L     41;
      T     #Robot_Prog_No;
_004: NOP   0;
      A     L      0.0;
      A     #M_BType_SP3;
      JNB   _005;
      L     51;
      T     #Robot_Prog_No;
_005: NOP   0;
NETWORK
TITLE =공정 차종 로보트 Program No.삭제

      AN    #M_BType_On;
      JNB   _006;
      L     0;
      T     #Robot_Prog_No;
_006: NOP   0;
END_FUNCTION_BLOCK

DATA_BLOCK DB 71
TITLE =
AUTHOR : SIMATIC
FAMILY : CPU_300
VERSION : 0.0

 FB 12
BEGIN
   REQ := FALSE;
   R := FALSE;
   ID := W#16#0;
   R_ID := DW#16#0;
   DONE := FALSE;
   ERROR := FALSE;
   STATUS := W#16#0;
   LEN := W#16#0;
   FB_ZUSTAND := B#16#0;
   REQ_SAVE := FALSE;
   R_SAVE := FALSE;
   ID_SAVE := W#16#0;
   R_ID_SAVE := DW#16#0;
   LEN_SAVE := W#16#0;
   SD_1_SAVE0 := W#16#0;
   SD_1_SAVE2 := W#16#0;
   SD_1_SAVE4 := W#16#0;
   SD_1_SAVE6 := W#16#0;
   SD_1_SAVE8 := W#16#0;
   HS_REQ_BYTE.rii := FALSE;
   HS_REQ_BYTE.nva := FALSE;
   HS_REQ_BYTE.ofs := FALSE;
   HS_REQ_BYTE.dir := FALSE;
   HS_REQ_BYTE.res := FALSE;
   HS_REQ_BYTE.roc := FALSE;
   HS_REQ_BYTE.nls := FALSE;
   HS_REQ_BYTE.rlo := FALSE;
   HS_RESP_BYTE.aii := FALSE;
   HS_RESP_BYTE.sns := FALSE;
   HS_RESP_BYTE.sqc := FALSE;
   HS_RESP_BYTE.ads := FALSE;
   HS_RESP_BYTE.aoc := FALSE;
   HS_RESP_BYTE.rs1 := FALSE;
   HS_RESP_BYTE.cnr := FALSE;
   HS_RESP_BYTE.rs2 := FALSE;
   HS_RESP_DSNR := B#16#0;
   HS_RESP_OFFSET := W#16#0;
   SD_1_WORD0 := W#16#0;
   SD_1_COUNT := W#16#0;
   SD_1_DBNUMMER := W#16#0;
   SD_1_DWORD6 := DW#16#0;
   SD_1_TYP := B#16#0;
   SFC_PARAM.LEN := W#16#0;
   SFC_PARAM.DB_NUMMER := W#16#0;
   SFC_PARAM.START := DW#16#0;
   BUFFER[0] := W#16#0;
   BUFFER[1] := W#16#0;
   BUFFER[2] := W#16#0;
   BUFFER[3] := W#16#0;
   BUFFER[4] := W#16#0;
   BUFFER[5] := W#16#0;
   BUFFER[6] := W#16#0;
   BUFFER[7] := W#16#0;
   BUFFER[8] := W#16#0;
   BUFFER[9] := W#16#0;
   BUFFER[10] := W#16#0;
   BUFFER[11] := W#16#0;
   BUFFER[12] := W#16#0;
   BUFFER[13] := W#16#0;
   BUFFER[14] := W#16#0;
   BUFFER[15] := W#16#0;
   BUFFER[16] := W#16#0;
   BUFFER[17] := W#16#0;
   BUFFER[18] := W#16#0;
   BUFFER[19] := W#16#0;
   BUFFER[20] := W#16#0;
   BUFFER[21] := W#16#0;
   BUFFER[22] := W#16#0;
   BUFFER[23] := W#16#0;
   BUFFER[24] := W#16#0;
   BUFFER[25] := W#16#0;
   BUFFER[26] := W#16#0;
   BUFFER[27] := W#16#0;
   BUFFER[28] := W#16#0;
   BUFFER[29] := W#16#0;
   BUFFER[30] := W#16#0;
   BUFFER[31] := W#16#0;
   BUFFER[32] := W#16#0;
   BUFFER[33] := W#16#0;
   BUFFER[34] := W#16#0;
   BUFFER[35] := W#16#0;
   BUFFER[36] := W#16#0;
   BUFFER[37] := W#16#0;
   BUFFER[38] := W#16#0;
   BUFFER[39] := W#16#0;
   BUFFER[40] := W#16#0;
   BUFFER[41] := W#16#0;
   BUFFER[42] := W#16#0;
   BUFFER[43] := W#16#0;
   BUFFER[44] := W#16#0;
   BUFFER[45] := W#16#0;
   BUFFER[46] := W#16#0;
   BUFFER[47] := W#16#0;
   BUFFER[48] := W#16#0;
   BUFFER[49] := W#16#0;
   BUFFER[50] := W#16#0;
   BUFFER[51] := W#16#0;
   BUFFER[52] := W#16#0;
   BUFFER[53] := W#16#0;
   BUFFER[54] := W#16#0;
   BUFFER[55] := W#16#0;
   BUFFER[56] := W#16#0;
   BUFFER[57] := W#16#0;
   BUFFER[58] := W#16#0;
   BUFFER[59] := W#16#0;
   BUFFER[60] := W#16#0;
   BUFFER[61] := W#16#0;
   BUFFER[62] := W#16#0;
   BUFFER[63] := W#16#0;
   BUFFER[64] := W#16#0;
   BUFFER[65] := W#16#0;
   BUFFER[66] := W#16#0;
   BUFFER[67] := W#16#0;
   BUFFER[68] := W#16#0;
   BUFFER[69] := W#16#0;
   BUFFER[70] := W#16#0;
   BUFFER[71] := W#16#0;
   BUFFER[72] := W#16#0;
   BUFFER[73] := W#16#0;
   BUFFER[74] := W#16#0;
   BUFFER[75] := W#16#0;
   BUFFER[76] := W#16#0;
   BUFFER[77] := W#16#0;
   BUFFER[78] := W#16#0;
   BUFFER[79] := W#16#0;
   BUFFER[80] := W#16#0;
   BUFFER[81] := W#16#0;
   BUFFER[82] := W#16#0;
   BUFFER[83] := W#16#0;
   BUFFER[84] := W#16#0;
   BUFFER[85] := W#16#0;
   BUFFER[86] := W#16#0;
   BUFFER[87] := W#16#0;
   BUFFER[88] := W#16#0;
   BUFFER[89] := W#16#0;
   BUFFER[90] := W#16#0;
   BUFFER[91] := W#16#0;
   BUFFER[92] := W#16#0;
   BUFFER[93] := W#16#0;
   BUFFER[94] := W#16#0;
   BUFFER[95] := W#16#0;
   BUFFER[96] := W#16#0;
   BUFFER[97] := W#16#0;
   BUFFER[98] := W#16#0;
   BUFFER[99] := W#16#0;
   BUFFER[100] := W#16#0;
   BUFFER[101] := W#16#0;
   BUFFER[102] := W#16#0;
   BUFFER[103] := W#16#0;
   BUFFER[104] := W#16#0;
   BUFFER[105] := W#16#0;
   BUFFER[106] := W#16#0;
   BUFFER[107] := W#16#0;
   BUFFER[108] := W#16#0;
   BUFFER[109] := W#16#0;
   BUFFER[110] := W#16#0;
   BUFFER[111] := W#16#0;
   BUFFER[112] := W#16#0;
   BUFFER[113] := W#16#0;
   BUFFER[114] := W#16#0;
   BUFFER[115] := W#16#0;
   BUFFER[116] := W#16#0;
   BUFFER[117] := W#16#0;
   BUFFER[118] := W#16#0;
   BUFFER[119] := W#16#0;
   REASON_FOR_CLOSE := B#16#0;
   DS_NR := B#16#0;
   PARAM_OFFSET := B#16#0;
   MAX_PUFF_LEN_SAVE := W#16#0;
   TYP_BOOL := FALSE;
   KANAL_PROBLEM := FALSE;
   KOMM_PROBLEM := FALSE;
   SEND_STARTED := FALSE;
   RECV_STARTED := FALSE;
   RESET_REQUEST := FALSE;
   RESET_EXECUTED := FALSE;
   DS200_BUSY := FALSE;
   MAX_DATA_LEN := W#16#0;
   LADDR_PTR := DW#16#0;
   FC_DATA_LEN := W#16#0;
   LADDR := W#16#0;
   SLEEP := B#16#0;
   SLEEP_EXT := B#16#0;
   ID_CLOSE := W#16#0;
   FB_KENNUNG := B#16#F1;
   RESERVE := B#16#0;
   ZUSTAND_WEICHE := B#16#0;
   SFB_AUFRUF.REQ := FALSE;
   SFB_AUFRUF.R := FALSE;
   SFB_AUFRUF.ID := W#16#0;
   SFB_AUFRUF.R_ID := DW#16#0;
   SFB_AUFRUF.DONE := FALSE;
   SFB_AUFRUF.ERROR := FALSE;
   SFB_AUFRUF.STATUS := W#16#0;
   SFB_AUFRUF.LEN := W#16#0;
   SFB_AUFRUF.INDEX := W#16#0;
   ZUSTAND_WEICHE_1 := B#16#0;
END_DATA_BLOCK

DATA_BLOCK DB 72
TITLE =
AUTHOR : SIMATIC
FAMILY : CPU_300
VERSION : 0.0

 FB 12
BEGIN
   REQ := FALSE;
   R := FALSE;
   ID := W#16#0;
   R_ID := DW#16#0;
   DONE := FALSE;
   ERROR := FALSE;
   STATUS := W#16#0;
   LEN := W#16#0;
   FB_ZUSTAND := B#16#0;
   REQ_SAVE := FALSE;
   R_SAVE := FALSE;
   ID_SAVE := W#16#0;
   R_ID_SAVE := DW#16#0;
   LEN_SAVE := W#16#0;
   SD_1_SAVE0 := W#16#0;
   SD_1_SAVE2 := W#16#0;
   SD_1_SAVE4 := W#16#0;
   SD_1_SAVE6 := W#16#0;
   SD_1_SAVE8 := W#16#0;
   HS_REQ_BYTE.rii := FALSE;
   HS_REQ_BYTE.nva := FALSE;
   HS_REQ_BYTE.ofs := FALSE;
   HS_REQ_BYTE.dir := FALSE;
   HS_REQ_BYTE.res := FALSE;
   HS_REQ_BYTE.roc := FALSE;
   HS_REQ_BYTE.nls := FALSE;
   HS_REQ_BYTE.rlo := FALSE;
   HS_RESP_BYTE.aii := FALSE;
   HS_RESP_BYTE.sns := FALSE;
   HS_RESP_BYTE.sqc := FALSE;
   HS_RESP_BYTE.ads := FALSE;
   HS_RESP_BYTE.aoc := FALSE;
   HS_RESP_BYTE.rs1 := FALSE;
   HS_RESP_BYTE.cnr := FALSE;
   HS_RESP_BYTE.rs2 := FALSE;
   HS_RESP_DSNR := B#16#0;
   HS_RESP_OFFSET := W#16#0;
   SD_1_WORD0 := W#16#0;
   SD_1_COUNT := W#16#0;
   SD_1_DBNUMMER := W#16#0;
   SD_1_DWORD6 := DW#16#0;
   SD_1_TYP := B#16#0;
   SFC_PARAM.LEN := W#16#0;
   SFC_PARAM.DB_NUMMER := W#16#0;
   SFC_PARAM.START := DW#16#0;
   BUFFER[0] := W#16#0;
   BUFFER[1] := W#16#0;
   BUFFER[2] := W#16#0;
   BUFFER[3] := W#16#0;
   BUFFER[4] := W#16#0;
   BUFFER[5] := W#16#0;
   BUFFER[6] := W#16#0;
   BUFFER[7] := W#16#0;
   BUFFER[8] := W#16#0;
   BUFFER[9] := W#16#0;
   BUFFER[10] := W#16#0;
   BUFFER[11] := W#16#0;
   BUFFER[12] := W#16#0;
   BUFFER[13] := W#16#0;
   BUFFER[14] := W#16#0;
   BUFFER[15] := W#16#0;
   BUFFER[16] := W#16#0;
   BUFFER[17] := W#16#0;
   BUFFER[18] := W#16#0;
   BUFFER[19] := W#16#0;
   BUFFER[20] := W#16#0;
   BUFFER[21] := W#16#0;
   BUFFER[22] := W#16#0;
   BUFFER[23] := W#16#0;
   BUFFER[24] := W#16#0;
   BUFFER[25] := W#16#0;
   BUFFER[26] := W#16#0;
   BUFFER[27] := W#16#0;
   BUFFER[28] := W#16#0;
   BUFFER[29] := W#16#0;
   BUFFER[30] := W#16#0;
   BUFFER[31] := W#16#0;
   BUFFER[32] := W#16#0;
   BUFFER[33] := W#16#0;
   BUFFER[34] := W#16#0;
   BUFFER[35] := W#16#0;
   BUFFER[36] := W#16#0;
   BUFFER[37] := W#16#0;
   BUFFER[38] := W#16#0;
   BUFFER[39] := W#16#0;
   BUFFER[40] := W#16#0;
   BUFFER[41] := W#16#0;
   BUFFER[42] := W#16#0;
   BUFFER[43] := W#16#0;
   BUFFER[44] := W#16#0;
   BUFFER[45] := W#16#0;
   BUFFER[46] := W#16#0;
   BUFFER[47] := W#16#0;
   BUFFER[48] := W#16#0;
   BUFFER[49] := W#16#0;
   BUFFER[50] := W#16#0;
   BUFFER[51] := W#16#0;
   BUFFER[52] := W#16#0;
   BUFFER[53] := W#16#0;
   BUFFER[54] := W#16#0;
   BUFFER[55] := W#16#0;
   BUFFER[56] := W#16#0;
   BUFFER[57] := W#16#0;
   BUFFER[58] := W#16#0;
   BUFFER[59] := W#16#0;
   BUFFER[60] := W#16#0;
   BUFFER[61] := W#16#0;
   BUFFER[62] := W#16#0;
   BUFFER[63] := W#16#0;
   BUFFER[64] := W#16#0;
   BUFFER[65] := W#16#0;
   BUFFER[66] := W#16#0;
   BUFFER[67] := W#16#0;
   BUFFER[68] := W#16#0;
   BUFFER[69] := W#16#0;
   BUFFER[70] := W#16#0;
   BUFFER[71] := W#16#0;
   BUFFER[72] := W#16#0;
   BUFFER[73] := W#16#0;
   BUFFER[74] := W#16#0;
   BUFFER[75] := W#16#0;
   BUFFER[76] := W#16#0;
   BUFFER[77] := W#16#0;
   BUFFER[78] := W#16#0;
   BUFFER[79] := W#16#0;
   BUFFER[80] := W#16#0;
   BUFFER[81] := W#16#0;
   BUFFER[82] := W#16#0;
   BUFFER[83] := W#16#0;
   BUFFER[84] := W#16#0;
   BUFFER[85] := W#16#0;
   BUFFER[86] := W#16#0;
   BUFFER[87] := W#16#0;
   BUFFER[88] := W#16#0;
   BUFFER[89] := W#16#0;
   BUFFER[90] := W#16#0;
   BUFFER[91] := W#16#0;
   BUFFER[92] := W#16#0;
   BUFFER[93] := W#16#0;
   BUFFER[94] := W#16#0;
   BUFFER[95] := W#16#0;
   BUFFER[96] := W#16#0;
   BUFFER[97] := W#16#0;
   BUFFER[98] := W#16#0;
   BUFFER[99] := W#16#0;
   BUFFER[100] := W#16#0;
   BUFFER[101] := W#16#0;
   BUFFER[102] := W#16#0;
   BUFFER[103] := W#16#0;
   BUFFER[104] := W#16#0;
   BUFFER[105] := W#16#0;
   BUFFER[106] := W#16#0;
   BUFFER[107] := W#16#0;
   BUFFER[108] := W#16#0;
   BUFFER[109] := W#16#0;
   BUFFER[110] := W#16#0;
   BUFFER[111] := W#16#0;
   BUFFER[112] := W#16#0;
   BUFFER[113] := W#16#0;
   BUFFER[114] := W#16#0;
   BUFFER[115] := W#16#0;
   BUFFER[116] := W#16#0;
   BUFFER[117] := W#16#0;
   BUFFER[118] := W#16#0;
   BUFFER[119] := W#16#0;
   REASON_FOR_CLOSE := B#16#0;
   DS_NR := B#16#0;
   PARAM_OFFSET := B#16#0;
   MAX_PUFF_LEN_SAVE := W#16#0;
   TYP_BOOL := FALSE;
   KANAL_PROBLEM := FALSE;
   KOMM_PROBLEM := FALSE;
   SEND_STARTED := FALSE;
   RECV_STARTED := FALSE;
   RESET_REQUEST := FALSE;
   RESET_EXECUTED := FALSE;
   DS200_BUSY := FALSE;
   MAX_DATA_LEN := W#16#0;
   LADDR_PTR := DW#16#0;
   FC_DATA_LEN := W#16#0;
   LADDR := W#16#0;
   SLEEP := B#16#0;
   SLEEP_EXT := B#16#0;
   ID_CLOSE := W#16#0;
   FB_KENNUNG := B#16#F1;
   RESERVE := B#16#0;
   ZUSTAND_WEICHE := B#16#0;
   SFB_AUFRUF.REQ := FALSE;
   SFB_AUFRUF.R := FALSE;
   SFB_AUFRUF.ID := W#16#0;
   SFB_AUFRUF.R_ID := DW#16#0;
   SFB_AUFRUF.DONE := FALSE;
   SFB_AUFRUF.ERROR := FALSE;
   SFB_AUFRUF.STATUS := W#16#0;
   SFB_AUFRUF.LEN := W#16#0;
   SFB_AUFRUF.INDEX := W#16#0;
   ZUSTAND_WEICHE_1 := B#16#0;
END_DATA_BLOCK

DATA_BLOCK DB 81
TITLE =
AUTHOR : SIMATIC
FAMILY : CPU_300
VERSION : 0.0

 FB 13
BEGIN
   EN_R := FALSE;
   ID := W#16#0;
   R_ID := DW#16#0;
   NDR := FALSE;
   ERROR := FALSE;
   STATUS := W#16#0;
   LEN := W#16#0;
   FB_ZUSTAND := B#16#0;
   EN_R_SAVE := FALSE;
   ID_SAVE := W#16#0;
   R_ID_SAVE := DW#16#0;
   FC_DATA_LEN := W#16#0;
   SD_1_SAVE0 := W#16#0;
   SD_1_SAVE2 := W#16#0;
   SD_1_SAVE4 := W#16#0;
   SD_1_SAVE6 := W#16#0;
   SD_1_SAVE8 := W#16#0;
   HS_REQ_BYTE.rii := FALSE;
   HS_REQ_BYTE.nva := FALSE;
   HS_REQ_BYTE.ofs := FALSE;
   HS_REQ_BYTE.dir := FALSE;
   HS_REQ_BYTE.res := FALSE;
   HS_REQ_BYTE.roc := FALSE;
   HS_REQ_BYTE.nls := FALSE;
   HS_REQ_BYTE.rlo := FALSE;
   HS_RESP_BYTE.aii := FALSE;
   HS_RESP_BYTE.sns := FALSE;
   HS_RESP_BYTE.sqc := FALSE;
   HS_RESP_BYTE.ads := FALSE;
   HS_RESP_BYTE.aoc := FALSE;
   HS_RESP_BYTE.rs1 := FALSE;
   HS_RESP_BYTE.cnr := FALSE;
   HS_RESP_BYTE.rs2 := FALSE;
   HS_RESP_DSNR := B#16#0;
   HS_RESP_OFFSET := W#16#0;
   SD_1_WORD0 := W#16#0;
   SD_1_COUNT := W#16#0;
   SD_1_DBNUMMER := W#16#0;
   SD_1_DWORD6 := DW#16#0;
   SD_1_TYP := B#16#0;
   SFC_PARAM.LEN := W#16#0;
   SFC_PARAM.DB_NUMMER := W#16#0;
   SFC_PARAM.START := DW#16#0;
   BUFFER[0] := W#16#0;
   BUFFER[1] := W#16#0;
   BUFFER[2] := W#16#0;
   BUFFER[3] := W#16#0;
   BUFFER[4] := W#16#0;
   BUFFER[5] := W#16#0;
   BUFFER[6] := W#16#0;
   BUFFER[7] := W#16#0;
   BUFFER[8] := W#16#0;
   BUFFER[9] := W#16#0;
   BUFFER[10] := W#16#0;
   BUFFER[11] := W#16#0;
   BUFFER[12] := W#16#0;
   BUFFER[13] := W#16#0;
   BUFFER[14] := W#16#0;
   BUFFER[15] := W#16#0;
   BUFFER[16] := W#16#0;
   BUFFER[17] := W#16#0;
   BUFFER[18] := W#16#0;
   BUFFER[19] := W#16#0;
   BUFFER[20] := W#16#0;
   BUFFER[21] := W#16#0;
   BUFFER[22] := W#16#0;
   BUFFER[23] := W#16#0;
   BUFFER[24] := W#16#0;
   BUFFER[25] := W#16#0;
   BUFFER[26] := W#16#0;
   BUFFER[27] := W#16#0;
   BUFFER[28] := W#16#0;
   BUFFER[29] := W#16#0;
   BUFFER[30] := W#16#0;
   BUFFER[31] := W#16#0;
   BUFFER[32] := W#16#0;
   BUFFER[33] := W#16#0;
   BUFFER[34] := W#16#0;
   BUFFER[35] := W#16#0;
   BUFFER[36] := W#16#0;
   BUFFER[37] := W#16#0;
   BUFFER[38] := W#16#0;
   BUFFER[39] := W#16#0;
   BUFFER[40] := W#16#0;
   BUFFER[41] := W#16#0;
   BUFFER[42] := W#16#0;
   BUFFER[43] := W#16#0;
   BUFFER[44] := W#16#0;
   BUFFER[45] := W#16#0;
   BUFFER[46] := W#16#0;
   BUFFER[47] := W#16#0;
   BUFFER[48] := W#16#0;
   BUFFER[49] := W#16#0;
   BUFFER[50] := W#16#0;
   BUFFER[51] := W#16#0;
   BUFFER[52] := W#16#0;
   BUFFER[53] := W#16#0;
   BUFFER[54] := W#16#0;
   BUFFER[55] := W#16#0;
   BUFFER[56] := W#16#0;
   BUFFER[57] := W#16#0;
   BUFFER[58] := W#16#0;
   BUFFER[59] := W#16#0;
   BUFFER[60] := W#16#0;
   BUFFER[61] := W#16#0;
   BUFFER[62] := W#16#0;
   BUFFER[63] := W#16#0;
   BUFFER[64] := W#16#0;
   BUFFER[65] := W#16#0;
   BUFFER[66] := W#16#0;
   BUFFER[67] := W#16#0;
   BUFFER[68] := W#16#0;
   BUFFER[69] := W#16#0;
   BUFFER[70] := W#16#0;
   BUFFER[71] := W#16#0;
   BUFFER[72] := W#16#0;
   BUFFER[73] := W#16#0;
   BUFFER[74] := W#16#0;
   BUFFER[75] := W#16#0;
   BUFFER[76] := W#16#0;
   BUFFER[77] := W#16#0;
   BUFFER[78] := W#16#0;
   BUFFER[79] := W#16#0;
   BUFFER[80] := W#16#0;
   BUFFER[81] := W#16#0;
   BUFFER[82] := W#16#0;
   BUFFER[83] := W#16#0;
   BUFFER[84] := W#16#0;
   BUFFER[85] := W#16#0;
   BUFFER[86] := W#16#0;
   BUFFER[87] := W#16#0;
   BUFFER[88] := W#16#0;
   BUFFER[89] := W#16#0;
   BUFFER[90] := W#16#0;
   BUFFER[91] := W#16#0;
   BUFFER[92] := W#16#0;
   BUFFER[93] := W#16#0;
   BUFFER[94] := W#16#0;
   BUFFER[95] := W#16#0;
   BUFFER[96] := W#16#0;
   BUFFER[97] := W#16#0;
   BUFFER[98] := W#16#0;
   BUFFER[99] := W#16#0;
   BUFFER[100] := W#16#0;
   BUFFER[101] := W#16#0;
   BUFFER[102] := W#16#0;
   BUFFER[103] := W#16#0;
   BUFFER[104] := W#16#0;
   BUFFER[105] := W#16#0;
   BUFFER[106] := W#16#0;
   BUFFER[107] := W#16#0;
   BUFFER[108] := W#16#0;
   BUFFER[109] := W#16#0;
   BUFFER[110] := W#16#0;
   BUFFER[111] := W#16#0;
   BUFFER[112] := W#16#0;
   BUFFER[113] := W#16#0;
   BUFFER[114] := W#16#0;
   BUFFER[115] := W#16#0;
   BUFFER[116] := W#16#0;
   BUFFER[117] := W#16#0;
   BUFFER[118] := W#16#0;
   BUFFER[119] := W#16#0;
   REASON_FOR_CLOSE := B#16#0;
   DS_NR := B#16#0;
   MAX_PUFF_LEN_SAVE := W#16#0;
   TYP_BOOL := FALSE;
   KANAL_PROBLEM := FALSE;
   KOMM_PROBLEM := FALSE;
   RECV_STARTED := FALSE;
   SEND_STARTED := FALSE;
   RESET_REQUEST := FALSE;
   RESET_EXECUTED := FALSE;
   DS200_BUSY := FALSE;
   LADDR_PTR := DW#16#0;
   LADDR := W#16#0;
   ZIEL_BYTE_SAVE := B#16#0;
   BOOL_ZIEL_BAD := FALSE;
   PARAM_OFFSET := DW#16#0;
   SLEEP := B#16#0;
   SLEEP_EXT := B#16#0;
   ID_CLOSE := W#16#0;
   RUNNING_LEN := W#16#0;
   FB_KENNUNG := B#16#F2;
   RESERVE := B#16#0;
   ZUSTAND_WEICHE := B#16#0;
   SFB_AUFRUF.EN_R := FALSE;
   SFB_AUFRUF.ID := W#16#0;
   SFB_AUFRUF.R_ID := DW#16#0;
   SFB_AUFRUF.NDR := FALSE;
   SFB_AUFRUF.ERROR := FALSE;
   SFB_AUFRUF.STATUS := W#16#0;
   SFB_AUFRUF.LEN := W#16#0;
   SFB_AUFRUF.INDEX := W#16#0;
   ZUSTAND_WEICHE_1 := B#16#0;
END_DATA_BLOCK

DATA_BLOCK DB 82
TITLE =
AUTHOR : SIMATIC
FAMILY : CPU_300
VERSION : 0.0

 FB 13
BEGIN
   EN_R := FALSE;
   ID := W#16#0;
   R_ID := DW#16#0;
   NDR := FALSE;
   ERROR := FALSE;
   STATUS := W#16#0;
   LEN := W#16#0;
   FB_ZUSTAND := B#16#0;
   EN_R_SAVE := FALSE;
   ID_SAVE := W#16#0;
   R_ID_SAVE := DW#16#0;
   FC_DATA_LEN := W#16#0;
   SD_1_SAVE0 := W#16#0;
   SD_1_SAVE2 := W#16#0;
   SD_1_SAVE4 := W#16#0;
   SD_1_SAVE6 := W#16#0;
   SD_1_SAVE8 := W#16#0;
   HS_REQ_BYTE.rii := FALSE;
   HS_REQ_BYTE.nva := FALSE;
   HS_REQ_BYTE.ofs := FALSE;
   HS_REQ_BYTE.dir := FALSE;
   HS_REQ_BYTE.res := FALSE;
   HS_REQ_BYTE.roc := FALSE;
   HS_REQ_BYTE.nls := FALSE;
   HS_REQ_BYTE.rlo := FALSE;
   HS_RESP_BYTE.aii := FALSE;
   HS_RESP_BYTE.sns := FALSE;
   HS_RESP_BYTE.sqc := FALSE;
   HS_RESP_BYTE.ads := FALSE;
   HS_RESP_BYTE.aoc := FALSE;
   HS_RESP_BYTE.rs1 := FALSE;
   HS_RESP_BYTE.cnr := FALSE;
   HS_RESP_BYTE.rs2 := FALSE;
   HS_RESP_DSNR := B#16#0;
   HS_RESP_OFFSET := W#16#0;
   SD_1_WORD0 := W#16#0;
   SD_1_COUNT := W#16#0;
   SD_1_DBNUMMER := W#16#0;
   SD_1_DWORD6 := DW#16#0;
   SD_1_TYP := B#16#0;
   SFC_PARAM.LEN := W#16#0;
   SFC_PARAM.DB_NUMMER := W#16#0;
   SFC_PARAM.START := DW#16#0;
   BUFFER[0] := W#16#0;
   BUFFER[1] := W#16#0;
   BUFFER[2] := W#16#0;
   BUFFER[3] := W#16#0;
   BUFFER[4] := W#16#0;
   BUFFER[5] := W#16#0;
   BUFFER[6] := W#16#0;
   BUFFER[7] := W#16#0;
   BUFFER[8] := W#16#0;
   BUFFER[9] := W#16#0;
   BUFFER[10] := W#16#0;
   BUFFER[11] := W#16#0;
   BUFFER[12] := W#16#0;
   BUFFER[13] := W#16#0;
   BUFFER[14] := W#16#0;
   BUFFER[15] := W#16#0;
   BUFFER[16] := W#16#0;
   BUFFER[17] := W#16#0;
   BUFFER[18] := W#16#0;
   BUFFER[19] := W#16#0;
   BUFFER[20] := W#16#0;
   BUFFER[21] := W#16#0;
   BUFFER[22] := W#16#0;
   BUFFER[23] := W#16#0;
   BUFFER[24] := W#16#0;
   BUFFER[25] := W#16#0;
   BUFFER[26] := W#16#0;
   BUFFER[27] := W#16#0;
   BUFFER[28] := W#16#0;
   BUFFER[29] := W#16#0;
   BUFFER[30] := W#16#0;
   BUFFER[31] := W#16#0;
   BUFFER[32] := W#16#0;
   BUFFER[33] := W#16#0;
   BUFFER[34] := W#16#0;
   BUFFER[35] := W#16#0;
   BUFFER[36] := W#16#0;
   BUFFER[37] := W#16#0;
   BUFFER[38] := W#16#0;
   BUFFER[39] := W#16#0;
   BUFFER[40] := W#16#0;
   BUFFER[41] := W#16#0;
   BUFFER[42] := W#16#0;
   BUFFER[43] := W#16#0;
   BUFFER[44] := W#16#0;
   BUFFER[45] := W#16#0;
   BUFFER[46] := W#16#0;
   BUFFER[47] := W#16#0;
   BUFFER[48] := W#16#0;
   BUFFER[49] := W#16#0;
   BUFFER[50] := W#16#0;
   BUFFER[51] := W#16#0;
   BUFFER[52] := W#16#0;
   BUFFER[53] := W#16#0;
   BUFFER[54] := W#16#0;
   BUFFER[55] := W#16#0;
   BUFFER[56] := W#16#0;
   BUFFER[57] := W#16#0;
   BUFFER[58] := W#16#0;
   BUFFER[59] := W#16#0;
   BUFFER[60] := W#16#0;
   BUFFER[61] := W#16#0;
   BUFFER[62] := W#16#0;
   BUFFER[63] := W#16#0;
   BUFFER[64] := W#16#0;
   BUFFER[65] := W#16#0;
   BUFFER[66] := W#16#0;
   BUFFER[67] := W#16#0;
   BUFFER[68] := W#16#0;
   BUFFER[69] := W#16#0;
   BUFFER[70] := W#16#0;
   BUFFER[71] := W#16#0;
   BUFFER[72] := W#16#0;
   BUFFER[73] := W#16#0;
   BUFFER[74] := W#16#0;
   BUFFER[75] := W#16#0;
   BUFFER[76] := W#16#0;
   BUFFER[77] := W#16#0;
   BUFFER[78] := W#16#0;
   BUFFER[79] := W#16#0;
   BUFFER[80] := W#16#0;
   BUFFER[81] := W#16#0;
   BUFFER[82] := W#16#0;
   BUFFER[83] := W#16#0;
   BUFFER[84] := W#16#0;
   BUFFER[85] := W#16#0;
   BUFFER[86] := W#16#0;
   BUFFER[87] := W#16#0;
   BUFFER[88] := W#16#0;
   BUFFER[89] := W#16#0;
   BUFFER[90] := W#16#0;
   BUFFER[91] := W#16#0;
   BUFFER[92] := W#16#0;
   BUFFER[93] := W#16#0;
   BUFFER[94] := W#16#0;
   BUFFER[95] := W#16#0;
   BUFFER[96] := W#16#0;
   BUFFER[97] := W#16#0;
   BUFFER[98] := W#16#0;
   BUFFER[99] := W#16#0;
   BUFFER[100] := W#16#0;
   BUFFER[101] := W#16#0;
   BUFFER[102] := W#16#0;
   BUFFER[103] := W#16#0;
   BUFFER[104] := W#16#0;
   BUFFER[105] := W#16#0;
   BUFFER[106] := W#16#0;
   BUFFER[107] := W#16#0;
   BUFFER[108] := W#16#0;
   BUFFER[109] := W#16#0;
   BUFFER[110] := W#16#0;
   BUFFER[111] := W#16#0;
   BUFFER[112] := W#16#0;
   BUFFER[113] := W#16#0;
   BUFFER[114] := W#16#0;
   BUFFER[115] := W#16#0;
   BUFFER[116] := W#16#0;
   BUFFER[117] := W#16#0;
   BUFFER[118] := W#16#0;
   BUFFER[119] := W#16#0;
   REASON_FOR_CLOSE := B#16#0;
   DS_NR := B#16#0;
   MAX_PUFF_LEN_SAVE := W#16#0;
   TYP_BOOL := FALSE;
   KANAL_PROBLEM := FALSE;
   KOMM_PROBLEM := FALSE;
   RECV_STARTED := FALSE;
   SEND_STARTED := FALSE;
   RESET_REQUEST := FALSE;
   RESET_EXECUTED := FALSE;
   DS200_BUSY := FALSE;
   LADDR_PTR := DW#16#0;
   LADDR := W#16#0;
   ZIEL_BYTE_SAVE := B#16#0;
   BOOL_ZIEL_BAD := FALSE;
   PARAM_OFFSET := DW#16#0;
   SLEEP := B#16#0;
   SLEEP_EXT := B#16#0;
   ID_CLOSE := W#16#0;
   RUNNING_LEN := W#16#0;
   FB_KENNUNG := B#16#F2;
   RESERVE := B#16#0;
   ZUSTAND_WEICHE := B#16#0;
   SFB_AUFRUF.EN_R := FALSE;
   SFB_AUFRUF.ID := W#16#0;
   SFB_AUFRUF.R_ID := DW#16#0;
   SFB_AUFRUF.NDR := FALSE;
   SFB_AUFRUF.ERROR := FALSE;
   SFB_AUFRUF.STATUS := W#16#0;
   SFB_AUFRUF.LEN := W#16#0;
   SFB_AUFRUF.INDEX := W#16#0;
   ZUSTAND_WEICHE_1 := B#16#0;
END_DATA_BLOCK

DATA_BLOCK DB 83
TITLE =
AUTHOR : SIMATIC
FAMILY : CPU_300
VERSION : 0.0

 FB 13
BEGIN
   EN_R := FALSE;
   ID := W#16#0;
   R_ID := DW#16#0;
   NDR := FALSE;
   ERROR := FALSE;
   STATUS := W#16#0;
   LEN := W#16#0;
   FB_ZUSTAND := B#16#0;
   EN_R_SAVE := FALSE;
   ID_SAVE := W#16#0;
   R_ID_SAVE := DW#16#0;
   FC_DATA_LEN := W#16#0;
   SD_1_SAVE0 := W#16#0;
   SD_1_SAVE2 := W#16#0;
   SD_1_SAVE4 := W#16#0;
   SD_1_SAVE6 := W#16#0;
   SD_1_SAVE8 := W#16#0;
   HS_REQ_BYTE.rii := FALSE;
   HS_REQ_BYTE.nva := FALSE;
   HS_REQ_BYTE.ofs := FALSE;
   HS_REQ_BYTE.dir := FALSE;
   HS_REQ_BYTE.res := FALSE;
   HS_REQ_BYTE.roc := FALSE;
   HS_REQ_BYTE.nls := FALSE;
   HS_REQ_BYTE.rlo := FALSE;
   HS_RESP_BYTE.aii := FALSE;
   HS_RESP_BYTE.sns := FALSE;
   HS_RESP_BYTE.sqc := FALSE;
   HS_RESP_BYTE.ads := FALSE;
   HS_RESP_BYTE.aoc := FALSE;
   HS_RESP_BYTE.rs1 := FALSE;
   HS_RESP_BYTE.cnr := FALSE;
   HS_RESP_BYTE.rs2 := FALSE;
   HS_RESP_DSNR := B#16#0;
   HS_RESP_OFFSET := W#16#0;
   SD_1_WORD0 := W#16#0;
   SD_1_COUNT := W#16#0;
   SD_1_DBNUMMER := W#16#0;
   SD_1_DWORD6 := DW#16#0;
   SD_1_TYP := B#16#0;
   SFC_PARAM.LEN := W#16#0;
   SFC_PARAM.DB_NUMMER := W#16#0;
   SFC_PARAM.START := DW#16#0;
   BUFFER[0] := W#16#0;
   BUFFER[1] := W#16#0;
   BUFFER[2] := W#16#0;
   BUFFER[3] := W#16#0;
   BUFFER[4] := W#16#0;
   BUFFER[5] := W#16#0;
   BUFFER[6] := W#16#0;
   BUFFER[7] := W#16#0;
   BUFFER[8] := W#16#0;
   BUFFER[9] := W#16#0;
   BUFFER[10] := W#16#0;
   BUFFER[11] := W#16#0;
   BUFFER[12] := W#16#0;
   BUFFER[13] := W#16#0;
   BUFFER[14] := W#16#0;
   BUFFER[15] := W#16#0;
   BUFFER[16] := W#16#0;
   BUFFER[17] := W#16#0;
   BUFFER[18] := W#16#0;
   BUFFER[19] := W#16#0;
   BUFFER[20] := W#16#0;
   BUFFER[21] := W#16#0;
   BUFFER[22] := W#16#0;
   BUFFER[23] := W#16#0;
   BUFFER[24] := W#16#0;
   BUFFER[25] := W#16#0;
   BUFFER[26] := W#16#0;
   BUFFER[27] := W#16#0;
   BUFFER[28] := W#16#0;
   BUFFER[29] := W#16#0;
   BUFFER[30] := W#16#0;
   BUFFER[31] := W#16#0;
   BUFFER[32] := W#16#0;
   BUFFER[33] := W#16#0;
   BUFFER[34] := W#16#0;
   BUFFER[35] := W#16#0;
   BUFFER[36] := W#16#0;
   BUFFER[37] := W#16#0;
   BUFFER[38] := W#16#0;
   BUFFER[39] := W#16#0;
   BUFFER[40] := W#16#0;
   BUFFER[41] := W#16#0;
   BUFFER[42] := W#16#0;
   BUFFER[43] := W#16#0;
   BUFFER[44] := W#16#0;
   BUFFER[45] := W#16#0;
   BUFFER[46] := W#16#0;
   BUFFER[47] := W#16#0;
   BUFFER[48] := W#16#0;
   BUFFER[49] := W#16#0;
   BUFFER[50] := W#16#0;
   BUFFER[51] := W#16#0;
   BUFFER[52] := W#16#0;
   BUFFER[53] := W#16#0;
   BUFFER[54] := W#16#0;
   BUFFER[55] := W#16#0;
   BUFFER[56] := W#16#0;
   BUFFER[57] := W#16#0;
   BUFFER[58] := W#16#0;
   BUFFER[59] := W#16#0;
   BUFFER[60] := W#16#0;
   BUFFER[61] := W#16#0;
   BUFFER[62] := W#16#0;
   BUFFER[63] := W#16#0;
   BUFFER[64] := W#16#0;
   BUFFER[65] := W#16#0;
   BUFFER[66] := W#16#0;
   BUFFER[67] := W#16#0;
   BUFFER[68] := W#16#0;
   BUFFER[69] := W#16#0;
   BUFFER[70] := W#16#0;
   BUFFER[71] := W#16#0;
   BUFFER[72] := W#16#0;
   BUFFER[73] := W#16#0;
   BUFFER[74] := W#16#0;
   BUFFER[75] := W#16#0;
   BUFFER[76] := W#16#0;
   BUFFER[77] := W#16#0;
   BUFFER[78] := W#16#0;
   BUFFER[79] := W#16#0;
   BUFFER[80] := W#16#0;
   BUFFER[81] := W#16#0;
   BUFFER[82] := W#16#0;
   BUFFER[83] := W#16#0;
   BUFFER[84] := W#16#0;
   BUFFER[85] := W#16#0;
   BUFFER[86] := W#16#0;
   BUFFER[87] := W#16#0;
   BUFFER[88] := W#16#0;
   BUFFER[89] := W#16#0;
   BUFFER[90] := W#16#0;
   BUFFER[91] := W#16#0;
   BUFFER[92] := W#16#0;
   BUFFER[93] := W#16#0;
   BUFFER[94] := W#16#0;
   BUFFER[95] := W#16#0;
   BUFFER[96] := W#16#0;
   BUFFER[97] := W#16#0;
   BUFFER[98] := W#16#0;
   BUFFER[99] := W#16#0;
   BUFFER[100] := W#16#0;
   BUFFER[101] := W#16#0;
   BUFFER[102] := W#16#0;
   BUFFER[103] := W#16#0;
   BUFFER[104] := W#16#0;
   BUFFER[105] := W#16#0;
   BUFFER[106] := W#16#0;
   BUFFER[107] := W#16#0;
   BUFFER[108] := W#16#0;
   BUFFER[109] := W#16#0;
   BUFFER[110] := W#16#0;
   BUFFER[111] := W#16#0;
   BUFFER[112] := W#16#0;
   BUFFER[113] := W#16#0;
   BUFFER[114] := W#16#0;
   BUFFER[115] := W#16#0;
   BUFFER[116] := W#16#0;
   BUFFER[117] := W#16#0;
   BUFFER[118] := W#16#0;
   BUFFER[119] := W#16#0;
   REASON_FOR_CLOSE := B#16#0;
   DS_NR := B#16#0;
   MAX_PUFF_LEN_SAVE := W#16#0;
   TYP_BOOL := FALSE;
   KANAL_PROBLEM := FALSE;
   KOMM_PROBLEM := FALSE;
   RECV_STARTED := FALSE;
   SEND_STARTED := FALSE;
   RESET_REQUEST := FALSE;
   RESET_EXECUTED := FALSE;
   DS200_BUSY := FALSE;
   LADDR_PTR := DW#16#0;
   LADDR := W#16#0;
   ZIEL_BYTE_SAVE := B#16#0;
   BOOL_ZIEL_BAD := FALSE;
   PARAM_OFFSET := DW#16#0;
   SLEEP := B#16#0;
   SLEEP_EXT := B#16#0;
   ID_CLOSE := W#16#0;
   RUNNING_LEN := W#16#0;
   FB_KENNUNG := B#16#F2;
   RESERVE := B#16#0;
   ZUSTAND_WEICHE := B#16#0;
   SFB_AUFRUF.EN_R := FALSE;
   SFB_AUFRUF.ID := W#16#0;
   SFB_AUFRUF.R_ID := DW#16#0;
   SFB_AUFRUF.NDR := FALSE;
   SFB_AUFRUF.ERROR := FALSE;
   SFB_AUFRUF.STATUS := W#16#0;
   SFB_AUFRUF.LEN := W#16#0;
   SFB_AUFRUF.INDEX := W#16#0;
   ZUSTAND_WEICHE_1 := B#16#0;
END_DATA_BLOCK

DATA_BLOCK DB 326
TITLE =
AUTHOR : ICom
FAMILY : DIAGNOSE
VERSION : 0.0

